//==========================================================
// 8) Extend automatic unload pulses
//==========================================================
// EN: A 500 ms pulse is compatible with integrated and third-party stackers.
// PT: Um pulso de 500 ms é compatível com stackers integrados e de terceiros.
instTPUpperStackerUnload(
    IN := upperStackerUnload,
    PT := T#500MS
);

instTPLowerStackerUnload(
    IN := lowerStackerUnload,
    PT := T#500MS
);

upperStackerUnload := instTPUpperStackerUnload.Q;
lowerStackerUnload := instTPLowerStackerUnload.Q;
END_ACTION

END_FUNCTION_BLOCK

// ---- POUs/MAIN.TcPOU
PROGRAM MAIN
VAR
	//==============================================================
	// EN: Main machine control function blocks
	// PT: Blocos principais de controle da máquina
	//==============================================================
	instFBSlitter1Control              : FB_SlitterControl;
	instFB_RotaryKnife                 : FB_RotaryKnife;
	// instFB_MetricsAndCalculation    : FB_MetricsAndCalculation;
	instFB_PaperDirectionControl       : FB_PaperDirectionControl;
	instFB_AutomaticOrderChange_V1     : FB_AutomaticOrderChange_V1;
	instFB_AlarmControl                : FB_AlarmControl;
	instFBSavePersistentData           : FB_SavePersistentData;

	//==============================================================
	// EN: Stacker control function blocks
	// PT: Blocos de controle dos empilhadores
	//==============================================================
	instFBLowerStackerControl          : FB_SimpleSheetStackerControl;
	instFBLowerStackerControlV1        : FB_SimpleSheetStackerControl_1;
	instFBUpperStackerControl          : FB_ComplexSheetStackerControl;

	//==============================================================
	// EN: Persistent data control status
	// PT: Estado do controle de dados persistentes
	//==============================================================
	bStart                             : BOOL;
	bError                             : BOOL;
	bBusy                              : BOOL;
	nErrorId                           : UDINT;
	fbR_Trig                           : R_TRIG;

	//==============================================================
	// EN: Machine interlock and control signals
	// PT: Sinais de intertravamento e controle da máquina
	//==============================================================
	slitterHomeComplete                : BOOL;
	aocReferenceSwitch                 : BOOL;
	lineSpeedUpFromAOC                 : BOOL;
	lineSpeedDownFromAOC               : BOOL;
	lineStopFromAOC                    : BOOL;
	executePositioningFromAOC          : BOOL;
	rotaryKnifeSpeedRefFromAOC         : LREAL;
	slitterSpeedRefFromAOC             : LREAL;
	lineStopFromRotaryKnife            : BOOL;
	lineStopFromSlitter                : BOOL;
	lineStopFromLowerStacker           : BOOL;
	aocRunning                         : BOOL;

	//==============================================================
	// EN: Program initialization
	// PT: Inicialização do programa
	//==============================================================
	firstScan                          : BOOL := TRUE;
	lineStopFromUpperStacker: BOOL;
END_VAR

//==============================================================
// EN: Cyclic machine control sequence
// PT: Sequência cíclica de controle da máquina
//==============================================================
_00_UpdateHardware();
_01_SlitterControl();
_02_RotaryKnifeControl();
_04_AutomaticOrderChange();
_05_LineControl();
_06_AlarmsControl();
_07_LowerStackerControl();
_08_UpperStackerControl();

// EN: Publish the upper stacker alarms and include them in the general indication.
// PT: Publica os alarmes do stacker superior e os inclui na indicação geral.
hmiAlarms.upperStacker :=
	instFBUpperStackerControl.hmiAlarms;

hmiStatus.alarmActive :=
	hmiStatus.alarmActive OR
	instFBUpperStackerControl.alarmActive;

// EN: Update persistent data management.
// PT: Atualiza o gerenciamento dos dados persistentes.
instFBSavePersistentData();

// EN: Apply default commands during the first PLC scan.
// PT: Aplica os comandos padrão durante o primeiro ciclo do PLC.
IF firstScan THEN
	hmiCommands.lowerStacker.backstopAutoCmd := TRUE;
	hmiCommands.lowerStacker.conveyorLevelerAutoCmd := TRUE;

	hmiCommands.upperStacker.backstopAutoCmd := TRUE;
	hmiCommands.upperStacker.elevatorAutoCmd := TRUE;

END_IF

firstScan := FALSE;

(*==============================================================================================================================
CPNTeck - Automação industrial
(c)Copyright 2023 All Rights Reserved
_______________________________________________________________________________________________________________________________
Library: <N/A or library name>
Tested with: <PLC / IPC model>
Engineering: <TwinCAT version>
Restrictions: <text>
Requirements: <text>
Functionality: <short description>
Support: <email>
Note: Parameter comments are only available in language 'English (United States)'
_______________________________________________________________________________________________________________________________
Change log table:

Version  		| Date        			| Expert in charge  	| Changes applied
<xx.xx.xx>		| <dd.mm.yyyy>  		| <name>              | <changes>

===============================================================================================================================*)

METHOD _00_UpdateHardware
VAR_INPUT
END_VAR

SLT1_P1_100_UG1();
SLT1_P1_100_UG2();
SLT1_P1_100_UG3();
SLT1_P1_100_UG4();
SLT1_P1_100_UG5();

SLT1_P1_200_UG1();
SLT1_P1_200_UG2();
SLT1_P1_200_UG3();
SLT1_P1_200_UG4();
SLT1_P1_200_UG5();
SLT1_P1_200_UG6();
SLT1_P1_200_UG7();
SLT1_P1_200_UG8();


STK_P2_050_DI1();
STK_P2_050_DI2();
STK_P2_050_DO1();
STK_P2_050_DO2();
	
STK_P2_050_AO1();	
STK_P2_050_AO2();
STK_P2_050_AO3();
STK_P2_050_AO4();

STK_P2_050_ENC1();
//Io-Link master
STK_050_BC2();
//Io-Link Slaves

STKU_050_DIO1();	//Ch 0 - IO-Link IP67 Input/Output module
STKU_050_DIO2(); //Ch 1 - IO-Link DIN Rail Input/Output module
STKU_050_DIO3(); //Ch 1 - IO-Link DIN Rail Input/Output module


STKL_050_DIO1();	//Ch 0 - IO-Link IP67 Input/Output module
STKL_050_DIO2(); //Ch 1 - IO-Link DIN Rail Input/Output module
STKL_100_B01(); //Ch 2 - IO-Link Pile height sensor	

//CANOpen slave	
STKU_P2_100_UG8(enable := TRUE); //Backstop servo drive

// EN: Lift servo drive. Quick stop is generated by the elevator control block.
// PT: Servo do elevador. O quick stop é gerado pelo bloco de controle do elevador.
STKU_P2_100_UG9(enable := TRUE);

// Safety processor (TwinSAFE)
STK_P2_050_SP01(run := TRUE,
				 errorAcknowledgement := hmiCommands.slitter1.resetCmd OR hmiCommands.lowerStacker.resetCmd OR hmiCommands.upperStacker.resetCmd,
				 safetyReset := hmiCommands.slitter1.resetCmd OR hmiCommands.lowerStacker.resetCmd OR hmiCommands.upperStacker.resetCmd
);
END_METHOD

METHOD _01_SlitterControl
VAR_INPUT
END_VAR

//ARK_P1_050_AO02.Channel1
//ARK_P1_050_AO02.Channel3
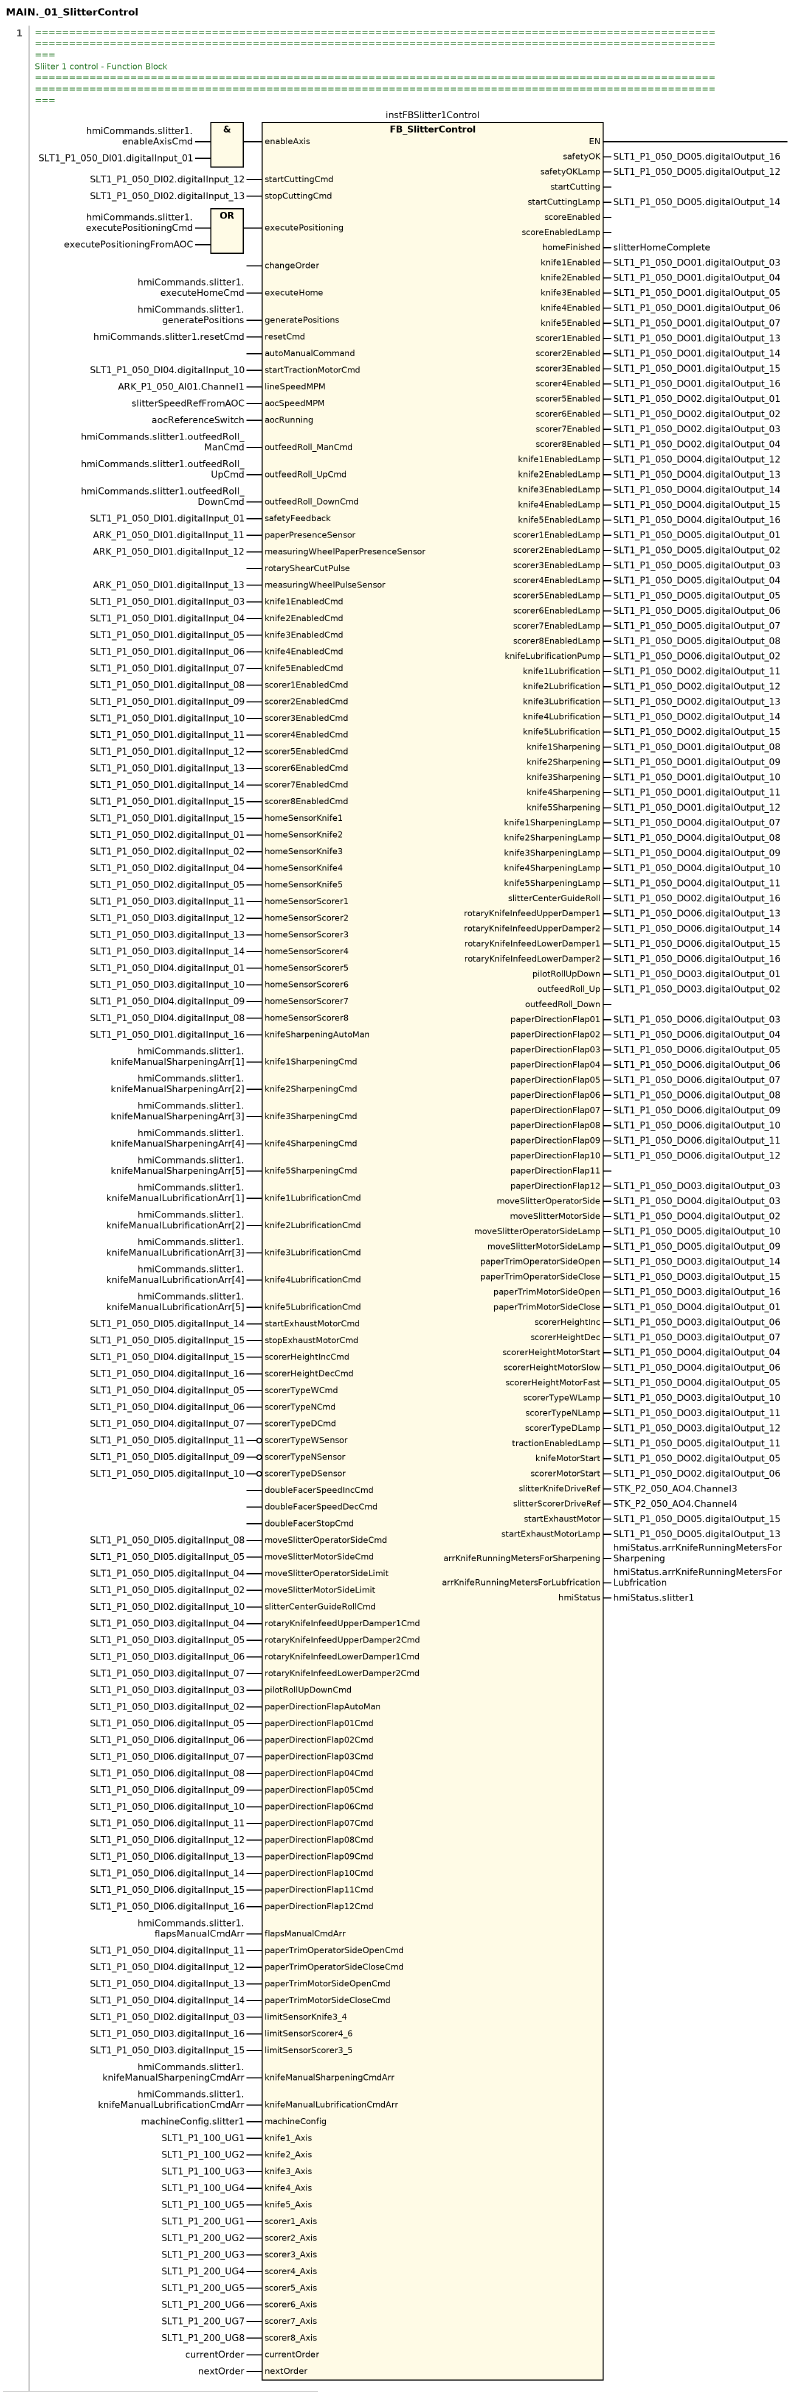
// NETWORK 1
// 					===========================================================================================================================================================================================================
//
// Sliiter 1 control - Function Block
//
// ===========================================================================================================================================================================================================
//
instFBSlitter1Control(
    enableAxis := hmiCommands.slitter1.enableAxisCmd AND SLT1_P1_050_DI01.digitalInput_01,
    startCuttingCmd := SLT1_P1_050_DI02.digitalInput_12,
    stopCuttingCmd := SLT1_P1_050_DI02.digitalInput_13,
    executePositioning := hmiCommands.slitter1.executePositioningCmd OR executePositioningFromAOC,
    executeHome := hmiCommands.slitter1.executeHomeCmd,
    generatePositions := hmiCommands.slitter1.generatePositions,
    resetCmd := hmiCommands.slitter1.resetCmd,
    startTractionMotorCmd := SLT1_P1_050_DI04.digitalInput_10,
    lineSpeedMPM := ARK_P1_050_AI01.Channel1,
    aocSpeedMPM := slitterSpeedRefFromAOC,
    aocRunning := aocReferenceSwitch,
    outfeedRoll_ManCmd := hmiCommands.slitter1.outfeedRoll_ManCmd,
    outfeedRoll_UpCmd := hmiCommands.slitter1.outfeedRoll_UpCmd,
    outfeedRoll_DownCmd := hmiCommands.slitter1.outfeedRoll_DownCmd,
    safetyFeedback := SLT1_P1_050_DI01.digitalInput_01,
    paperPresenceSensor := ARK_P1_050_DI01.digitalInput_11,
    measuringWheelPaperPresenceSensor := ARK_P1_050_DI01.digitalInput_12,
    measuringWheelPulseSensor := ARK_P1_050_DI01.digitalInput_13,
    knife1EnabledCmd := SLT1_P1_050_DI01.digitalInput_03,
    knife2EnabledCmd := SLT1_P1_050_DI01.digitalInput_04,
    knife3EnabledCmd := SLT1_P1_050_DI01.digitalInput_05,
    knife4EnabledCmd := SLT1_P1_050_DI01.digitalInput_06,
    knife5EnabledCmd := SLT1_P1_050_DI01.digitalInput_07,
    scorer1EnabledCmd := SLT1_P1_050_DI01.digitalInput_08,
    scorer2EnabledCmd := SLT1_P1_050_DI01.digitalInput_09,
    scorer3EnabledCmd := SLT1_P1_050_DI01.digitalInput_10,
    scorer4EnabledCmd := SLT1_P1_050_DI01.digitalInput_11,
    scorer5EnabledCmd := SLT1_P1_050_DI01.digitalInput_12,
    scorer6EnabledCmd := SLT1_P1_050_DI01.digitalInput_13,
    scorer7EnabledCmd := SLT1_P1_050_DI01.digitalInput_14,
    scorer8EnabledCmd := SLT1_P1_050_DI01.digitalInput_15,
    homeSensorKnife1 := SLT1_P1_050_DI01.digitalInput_15,
    homeSensorKnife2 := SLT1_P1_050_DI02.digitalInput_01,
    homeSensorKnife3 := SLT1_P1_050_DI02.digitalInput_02,
    homeSensorKnife4 := SLT1_P1_050_DI02.digitalInput_04,
    homeSensorKnife5 := SLT1_P1_050_DI02.digitalInput_05,
    homeSensorScorer1 := SLT1_P1_050_DI03.digitalInput_11,
    homeSensorScorer2 := SLT1_P1_050_DI03.digitalInput_12,
    homeSensorScorer3 := SLT1_P1_050_DI03.digitalInput_13,
    homeSensorScorer4 := SLT1_P1_050_DI03.digitalInput_14,
    homeSensorScorer5 := SLT1_P1_050_DI04.digitalInput_01,
    homeSensorScorer6 := SLT1_P1_050_DI03.digitalInput_10,
    homeSensorScorer7 := SLT1_P1_050_DI04.digitalInput_09,
    homeSensorScorer8 := SLT1_P1_050_DI04.digitalInput_08,
    knifeSharpeningAutoMan := SLT1_P1_050_DI01.digitalInput_16,
    knife1SharpeningCmd := hmiCommands.slitter1.knifeManualSharpeningArr[1],
    knife2SharpeningCmd := hmiCommands.slitter1.knifeManualSharpeningArr[2],
    knife3SharpeningCmd := hmiCommands.slitter1.knifeManualSharpeningArr[3],
    knife4SharpeningCmd := hmiCommands.slitter1.knifeManualSharpeningArr[4],
    knife5SharpeningCmd := hmiCommands.slitter1.knifeManualSharpeningArr[5],
    knife1LubrificationCmd := hmiCommands.slitter1.knifeManualLubrificationArr[1],
    knife2LubrificationCmd := hmiCommands.slitter1.knifeManualLubrificationArr[2],
    knife3LubrificationCmd := hmiCommands.slitter1.knifeManualLubrificationArr[3],
    knife4LubrificationCmd := hmiCommands.slitter1.knifeManualLubrificationArr[4],
    knife5LubrificationCmd := hmiCommands.slitter1.knifeManualLubrificationArr[5],
    startExhaustMotorCmd := SLT1_P1_050_DI05.digitalInput_14,
    stopExhaustMotorCmd := SLT1_P1_050_DI05.digitalInput_15,
    scorerHeightIncCmd := SLT1_P1_050_DI04.digitalInput_15,
    scorerHeightDecCmd := SLT1_P1_050_DI04.digitalInput_16,
    scorerTypeWCmd := SLT1_P1_050_DI04.digitalInput_05,
    scorerTypeNCmd := SLT1_P1_050_DI04.digitalInput_06,
    scorerTypeDCmd := SLT1_P1_050_DI04.digitalInput_07,
    scorerTypeWSensor := NOT SLT1_P1_050_DI05.digitalInput_11,
    scorerTypeNSensor := NOT SLT1_P1_050_DI05.digitalInput_09,
    scorerTypeDSensor := NOT SLT1_P1_050_DI05.digitalInput_10,
    moveSlitterOperatorSideCmd := SLT1_P1_050_DI05.digitalInput_08,
    moveSlitterMotorSideCmd := SLT1_P1_050_DI05.digitalInput_05,
    moveSlitterOperatorSideLimit := SLT1_P1_050_DI05.digitalInput_04,
    moveSlitterMotorSideLimit := SLT1_P1_050_DI05.digitalInput_02,
    slitterCenterGuideRollCmd := SLT1_P1_050_DI02.digitalInput_10,
    rotaryKnifeInfeedUpperDamper1Cmd := SLT1_P1_050_DI03.digitalInput_04,
    rotaryKnifeInfeedUpperDamper2Cmd := SLT1_P1_050_DI03.digitalInput_05,
    rotaryKnifeInfeedLowerDamper1Cmd := SLT1_P1_050_DI03.digitalInput_06,
    rotaryKnifeInfeedLowerDamper2Cmd := SLT1_P1_050_DI03.digitalInput_07,
    pilotRollUpDownCmd := SLT1_P1_050_DI03.digitalInput_03,
    paperDirectionFlapAutoMan := SLT1_P1_050_DI03.digitalInput_02,
    paperDirectionFlap01Cmd := SLT1_P1_050_DI06.digitalInput_05,
    paperDirectionFlap02Cmd := SLT1_P1_050_DI06.digitalInput_06,
    paperDirectionFlap03Cmd := SLT1_P1_050_DI06.digitalInput_07,
    paperDirectionFlap04Cmd := SLT1_P1_050_DI06.digitalInput_08,
    paperDirectionFlap05Cmd := SLT1_P1_050_DI06.digitalInput_09,
    paperDirectionFlap06Cmd := SLT1_P1_050_DI06.digitalInput_10,
    paperDirectionFlap07Cmd := SLT1_P1_050_DI06.digitalInput_11,
    paperDirectionFlap08Cmd := SLT1_P1_050_DI06.digitalInput_12,
    paperDirectionFlap09Cmd := SLT1_P1_050_DI06.digitalInput_13,
    paperDirectionFlap10Cmd := SLT1_P1_050_DI06.digitalInput_14,
    paperDirectionFlap11Cmd := SLT1_P1_050_DI06.digitalInput_15,
    paperDirectionFlap12Cmd := SLT1_P1_050_DI06.digitalInput_16,
    flapsManualCmdArr := hmiCommands.slitter1.flapsManualCmdArr,
    paperTrimOperatorSideOpenCmd := SLT1_P1_050_DI04.digitalInput_11,
    paperTrimOperatorSideCloseCmd := SLT1_P1_050_DI04.digitalInput_12,
    paperTrimMotorSideOpenCmd := SLT1_P1_050_DI04.digitalInput_13,
    paperTrimMotorSideCloseCmd := SLT1_P1_050_DI04.digitalInput_14,
    limitSensorKnife3_4 := SLT1_P1_050_DI02.digitalInput_03,
    limitSensorScorer4_6 := SLT1_P1_050_DI03.digitalInput_16,
    limitSensorScorer3_5 := SLT1_P1_050_DI03.digitalInput_15,
    knifeManualSharpeningCmdArr := hmiCommands.slitter1.knifeManualSharpeningCmdArr,
    knifeManualLubrificationCmdArr := hmiCommands.slitter1.knifeManualLubrificationCmdArr,
    machineConfig := machineConfig.slitter1,
    knife1_Axis := SLT1_P1_100_UG1,
    knife2_Axis := SLT1_P1_100_UG2,
    knife3_Axis := SLT1_P1_100_UG3,
    knife4_Axis := SLT1_P1_100_UG4,
    knife5_Axis := SLT1_P1_100_UG5,
    scorer1_Axis := SLT1_P1_200_UG1,
    scorer2_Axis := SLT1_P1_200_UG2,
    scorer3_Axis := SLT1_P1_200_UG3,
    scorer4_Axis := SLT1_P1_200_UG4,
    scorer5_Axis := SLT1_P1_200_UG5,
    scorer6_Axis := SLT1_P1_200_UG6,
    scorer7_Axis := SLT1_P1_200_UG7,
    scorer8_Axis := SLT1_P1_200_UG8,
    currentOrder := currentOrder,
    nextOrder := nextOrder,
    safetyOK => SLT1_P1_050_DO05.digitalOutput_16,
    safetyOKLamp => SLT1_P1_050_DO05.digitalOutput_12,
    startCuttingLamp => SLT1_P1_050_DO05.digitalOutput_14,
    homeFinished => slitterHomeComplete,
    knife1Enabled => SLT1_P1_050_DO01.digitalOutput_03,
    knife2Enabled => SLT1_P1_050_DO01.digitalOutput_04,
    knife3Enabled => SLT1_P1_050_DO01.digitalOutput_05,
    knife4Enabled => SLT1_P1_050_DO01.digitalOutput_06,
    knife5Enabled => SLT1_P1_050_DO01.digitalOutput_07,
    scorer1Enabled => SLT1_P1_050_DO01.digitalOutput_13,
    scorer2Enabled => SLT1_P1_050_DO01.digitalOutput_14,
    scorer3Enabled => SLT1_P1_050_DO01.digitalOutput_15,
    scorer4Enabled => SLT1_P1_050_DO01.digitalOutput_16,
    scorer5Enabled => SLT1_P1_050_DO02.digitalOutput_01,
    scorer6Enabled => SLT1_P1_050_DO02.digitalOutput_02,
    scorer7Enabled => SLT1_P1_050_DO02.digitalOutput_03,
    scorer8Enabled => SLT1_P1_050_DO02.digitalOutput_04,
    knife1EnabledLamp => SLT1_P1_050_DO04.digitalOutput_12,
    knife2EnabledLamp => SLT1_P1_050_DO04.digitalOutput_13,
    knife3EnabledLamp => SLT1_P1_050_DO04.digitalOutput_14,
    knife4EnabledLamp => SLT1_P1_050_DO04.digitalOutput_15,
    knife5EnabledLamp => SLT1_P1_050_DO04.digitalOutput_16,
    scorer1EnabledLamp => SLT1_P1_050_DO05.digitalOutput_01,
    scorer2EnabledLamp => SLT1_P1_050_DO05.digitalOutput_02,
    scorer3EnabledLamp => SLT1_P1_050_DO05.digitalOutput_03,
    scorer4EnabledLamp => SLT1_P1_050_DO05.digitalOutput_04,
    scorer5EnabledLamp => SLT1_P1_050_DO05.digitalOutput_05,
    scorer6EnabledLamp => SLT1_P1_050_DO05.digitalOutput_06,
    scorer7EnabledLamp => SLT1_P1_050_DO05.digitalOutput_07,
    scorer8EnabledLamp => SLT1_P1_050_DO05.digitalOutput_08,
    knifeLubrificationPump => SLT1_P1_050_DO06.digitalOutput_02,
    knife1Lubrification => SLT1_P1_050_DO02.digitalOutput_11,
    knife2Lubrification => SLT1_P1_050_DO02.digitalOutput_12,
    knife3Lubrification => SLT1_P1_050_DO02.digitalOutput_13,
    knife4Lubrification => SLT1_P1_050_DO02.digitalOutput_14,
    knife5Lubrification => SLT1_P1_050_DO02.digitalOutput_15,
    knife1Sharpening => SLT1_P1_050_DO01.digitalOutput_08,
    knife2Sharpening => SLT1_P1_050_DO01.digitalOutput_09,
    knife3Sharpening => SLT1_P1_050_DO01.digitalOutput_10,
    knife4Sharpening => SLT1_P1_050_DO01.digitalOutput_11,
    knife5Sharpening => SLT1_P1_050_DO01.digitalOutput_12,
    knife1SharpeningLamp => SLT1_P1_050_DO04.digitalOutput_07,
    knife2SharpeningLamp => SLT1_P1_050_DO04.digitalOutput_08,
    knife3SharpeningLamp => SLT1_P1_050_DO04.digitalOutput_09,
    knife4SharpeningLamp => SLT1_P1_050_DO04.digitalOutput_10,
    knife5SharpeningLamp => SLT1_P1_050_DO04.digitalOutput_11,
    slitterCenterGuideRoll => SLT1_P1_050_DO02.digitalOutput_16,
    rotaryKnifeInfeedUpperDamper1 => SLT1_P1_050_DO06.digitalOutput_13,
    rotaryKnifeInfeedUpperDamper2 => SLT1_P1_050_DO06.digitalOutput_14,
    rotaryKnifeInfeedLowerDamper1 => SLT1_P1_050_DO06.digitalOutput_15,
    rotaryKnifeInfeedLowerDamper2 => SLT1_P1_050_DO06.digitalOutput_16,
    pilotRollUpDown => SLT1_P1_050_DO03.digitalOutput_01,
    outfeedRoll_Up => SLT1_P1_050_DO03.digitalOutput_02,
    paperDirectionFlap01 => SLT1_P1_050_DO06.digitalOutput_03,
    paperDirectionFlap02 => SLT1_P1_050_DO06.digitalOutput_04,
    paperDirectionFlap03 => SLT1_P1_050_DO06.digitalOutput_05,
    paperDirectionFlap04 => SLT1_P1_050_DO06.digitalOutput_06,
    paperDirectionFlap05 => SLT1_P1_050_DO06.digitalOutput_07,
    paperDirectionFlap06 => SLT1_P1_050_DO06.digitalOutput_08,
    paperDirectionFlap07 => SLT1_P1_050_DO06.digitalOutput_09,
    paperDirectionFlap08 => SLT1_P1_050_DO06.digitalOutput_10,
    paperDirectionFlap09 => SLT1_P1_050_DO06.digitalOutput_11,
    paperDirectionFlap10 => SLT1_P1_050_DO06.digitalOutput_12,
    paperDirectionFlap12 => SLT1_P1_050_DO03.digitalOutput_03,
    moveSlitterOperatorSide => SLT1_P1_050_DO04.digitalOutput_03,
    moveSlitterMotorSide => SLT1_P1_050_DO04.digitalOutput_02,
    moveSlitterOperatorSideLamp => SLT1_P1_050_DO05.digitalOutput_10,
    moveSlitterMotorSideLamp => SLT1_P1_050_DO05.digitalOutput_09,
    paperTrimOperatorSideOpen => SLT1_P1_050_DO03.digitalOutput_14,
    paperTrimOperatorSideClose => SLT1_P1_050_DO03.digitalOutput_15,
    paperTrimMotorSideOpen => SLT1_P1_050_DO03.digitalOutput_16,
    paperTrimMotorSideClose => SLT1_P1_050_DO04.digitalOutput_01,
    scorerHeightInc => SLT1_P1_050_DO03.digitalOutput_06,
    scorerHeightDec => SLT1_P1_050_DO03.digitalOutput_07,
    scorerHeightMotorStart => SLT1_P1_050_DO04.digitalOutput_04,
    scorerHeightMotorSlow => SLT1_P1_050_DO04.digitalOutput_06,
    scorerHeightMotorFast => SLT1_P1_050_DO04.digitalOutput_05,
    scorerTypeWLamp => SLT1_P1_050_DO03.digitalOutput_10,
    scorerTypeNLamp => SLT1_P1_050_DO03.digitalOutput_11,
    scorerTypeDLamp => SLT1_P1_050_DO03.digitalOutput_12,
    tractionEnabledLamp => SLT1_P1_050_DO05.digitalOutput_11,
    knifeMotorStart => SLT1_P1_050_DO02.digitalOutput_05,
    scorerMotorStart => SLT1_P1_050_DO02.digitalOutput_06,
    slitterKnifeDriveRef => STK_P2_050_AO4.Channel3,
    slitterScorerDriveRef => STK_P2_050_AO4.Channel4,
    startExhaustMotor => SLT1_P1_050_DO05.digitalOutput_15,
    startExhaustMotorLamp => SLT1_P1_050_DO05.digitalOutput_13,
    arrKnifeRunningMetersForSharpening => hmiStatus.arrKnifeRunningMetersForSharpening,
    arrKnifeRunningMetersForLubfrication => hmiStatus.arrKnifeRunningMetersForLubfrication,
    hmiStatus => hmiStatus.slitter1); // FB_SlitterControl
END_METHOD

METHOD _02_RotaryKnifeControl
VAR_INPUT
END_VAR

(*


ARK_050_DI01.digitalInput_01 => exitGuardOpen
ARK_050_DI01.digitalInput_02 => lowerKnifeGuardClosed
ARK_050_DI01.digitalInput_03 => upperKnifeGuardClosed
ARK_050_DI01.digitalInput_04 => infeedGuardOpen

ARK_050_DI01.digitalInput_05 => lowerOilLevelLow
ARK_050_DI01.digitalInput_06 => upperOilLevelLow
ARK_050_DI01.digitalInput_07 => exhaustPressurized
ARK_050_DI01.digitalInput_08 => exhaustDepressurized

ARK_050_DI01.digitalInput_09 => upperLevelPaperSensor
ARK_050_DI01.digitalInput_10 => upperKnifeJamDetected
ARK_050_DI01.digitalInput_11 => lowerLevelPaperSensor
ARK_050_DI01.digitalInput_12 => lowerKnifeJamDetected

ARK_050_DI01.digitalInput_13 => lowerKnifeHome
ARK_050_DI01.digitalInput_14 => upperKnifeHome

*)
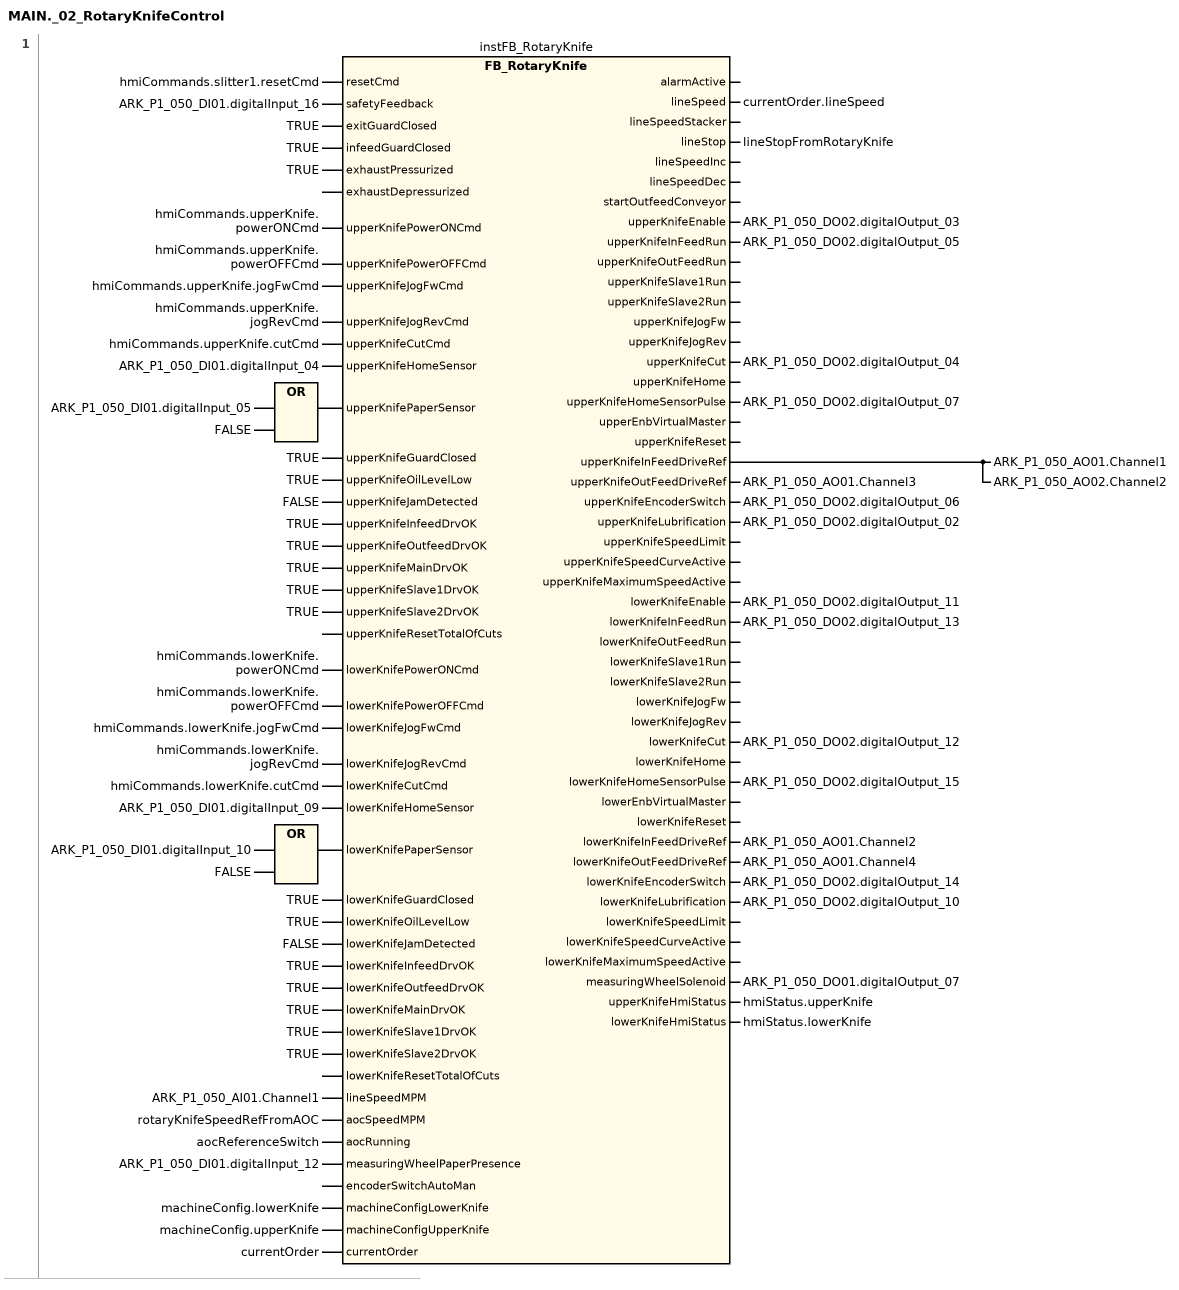
// NETWORK 1
instFB_RotaryKnife(
    resetCmd := hmiCommands.slitter1.resetCmd,
    safetyFeedback := ARK_P1_050_DI01.digitalInput_16,
    exitGuardClosed := TRUE,
    infeedGuardClosed := TRUE,
    exhaustPressurized := TRUE,
    upperKnifePowerONCmd := hmiCommands.upperKnife.powerONCmd,
    upperKnifePowerOFFCmd := hmiCommands.upperKnife.powerOFFCmd,
    upperKnifeJogFwCmd := hmiCommands.upperKnife.jogFwCmd,
    upperKnifeJogRevCmd := hmiCommands.upperKnife.jogRevCmd,
    upperKnifeCutCmd := hmiCommands.upperKnife.cutCmd,
    upperKnifeHomeSensor := ARK_P1_050_DI01.digitalInput_04,
    upperKnifePaperSensor := ARK_P1_050_DI01.digitalInput_05 OR FALSE,
    upperKnifeGuardClosed := TRUE,
    upperKnifeOilLevelLow := TRUE,
    upperKnifeJamDetected := FALSE,
    upperKnifeInfeedDrvOK := TRUE,
    upperKnifeOutfeedDrvOK := TRUE,
    upperKnifeMainDrvOK := TRUE,
    upperKnifeSlave1DrvOK := TRUE,
    upperKnifeSlave2DrvOK := TRUE,
    lowerKnifePowerONCmd := hmiCommands.lowerKnife.powerONCmd,
    lowerKnifePowerOFFCmd := hmiCommands.lowerKnife.powerOFFCmd,
    lowerKnifeJogFwCmd := hmiCommands.lowerKnife.jogFwCmd,
    lowerKnifeJogRevCmd := hmiCommands.lowerKnife.jogRevCmd,
    lowerKnifeCutCmd := hmiCommands.lowerKnife.cutCmd,
    lowerKnifeHomeSensor := ARK_P1_050_DI01.digitalInput_09,
    lowerKnifePaperSensor := ARK_P1_050_DI01.digitalInput_10 OR FALSE,
    lowerKnifeGuardClosed := TRUE,
    lowerKnifeOilLevelLow := TRUE,
    lowerKnifeJamDetected := FALSE,
    lowerKnifeInfeedDrvOK := TRUE,
    lowerKnifeOutfeedDrvOK := TRUE,
    lowerKnifeMainDrvOK := TRUE,
    lowerKnifeSlave1DrvOK := TRUE,
    lowerKnifeSlave2DrvOK := TRUE,
    lineSpeedMPM := ARK_P1_050_AI01.Channel1,
    aocSpeedMPM := rotaryKnifeSpeedRefFromAOC,
    aocRunning := aocReferenceSwitch,
    measuringWheelPaperPresence := ARK_P1_050_DI01.digitalInput_12,
    machineConfigLowerKnife := machineConfig.lowerKnife,
    machineConfigUpperKnife := machineConfig.upperKnife,
    currentOrder := currentOrder,
    lineSpeed => currentOrder.lineSpeed,
    lineStop => lineStopFromRotaryKnife,
    upperKnifeEnable => ARK_P1_050_DO02.digitalOutput_03,
    upperKnifeInFeedRun => ARK_P1_050_DO02.digitalOutput_05,
    upperKnifeCut => ARK_P1_050_DO02.digitalOutput_04,
    upperKnifeHomeSensorPulse => ARK_P1_050_DO02.digitalOutput_07,
    upperKnifeOutFeedDriveRef => ARK_P1_050_AO01.Channel3,
    upperKnifeEncoderSwitch => ARK_P1_050_DO02.digitalOutput_06,
    upperKnifeLubrification => ARK_P1_050_DO02.digitalOutput_02,
    lowerKnifeEnable => ARK_P1_050_DO02.digitalOutput_11,
    lowerKnifeInFeedRun => ARK_P1_050_DO02.digitalOutput_13,
    lowerKnifeCut => ARK_P1_050_DO02.digitalOutput_12,
    lowerKnifeHomeSensorPulse => ARK_P1_050_DO02.digitalOutput_15,
    lowerKnifeInFeedDriveRef => ARK_P1_050_AO01.Channel2,
    lowerKnifeOutFeedDriveRef => ARK_P1_050_AO01.Channel4,
    lowerKnifeEncoderSwitch => ARK_P1_050_DO02.digitalOutput_14,
    lowerKnifeLubrification => ARK_P1_050_DO02.digitalOutput_10,
    measuringWheelSolenoid => ARK_P1_050_DO01.digitalOutput_07,
    upperKnifeHmiStatus => hmiStatus.upperKnife,
    lowerKnifeHmiStatus => hmiStatus.lowerKnife); // FB_RotaryKnife
ARK_P1_050_AO01.Channel1 := instFB_RotaryKnife.upperKnifeInFeedDriveRef;
ARK_P1_050_AO02.Channel2 := instFB_RotaryKnife.upperKnifeInFeedDriveRef;
END_METHOD

METHOD _04_AutomaticOrderChange
VAR_INPUT
END_VAR
(*

	SLT1_C1_050_DI01     : FB_EL1809;        // Digital inputs card
    SLT1_C1_050_DO01     : FB_EL2809;        // Digital outputs card

*)
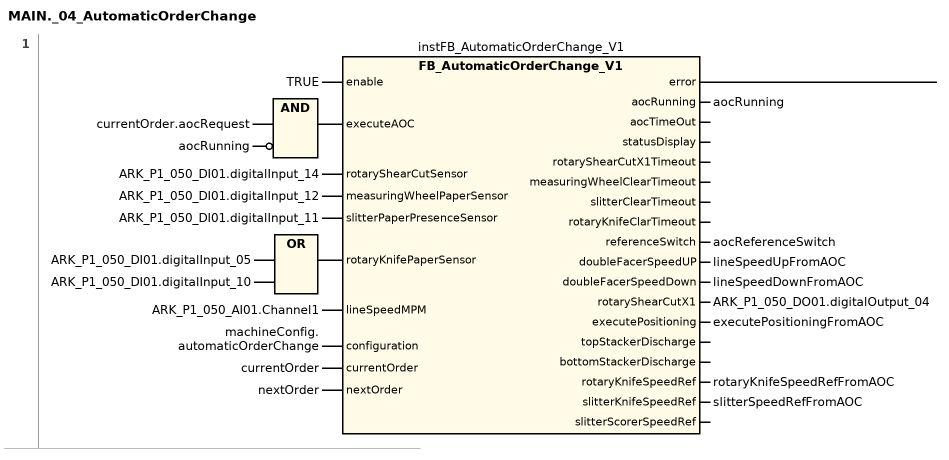
// NETWORK 1
instFB_AutomaticOrderChange_V1(
    enable := TRUE,
    executeAOC := currentOrder.aocRequest AND NOT aocRunning,
    rotaryShearCutSensor := ARK_P1_050_DI01.digitalInput_14,
    measuringWheelPaperSensor := ARK_P1_050_DI01.digitalInput_12,
    slitterPaperPresenceSensor := ARK_P1_050_DI01.digitalInput_11,
    rotaryKnifePaperSensor := ARK_P1_050_DI01.digitalInput_05 OR ARK_P1_050_DI01.digitalInput_10,
    lineSpeedMPM := ARK_P1_050_AI01.Channel1,
    configuration := machineConfig.automaticOrderChange,
    currentOrder := currentOrder,
    nextOrder := nextOrder,
    aocRunning => aocRunning,
    referenceSwitch => aocReferenceSwitch,
    doubleFacerSpeedUP => lineSpeedUpFromAOC,
    doubleFacerSpeedDown => lineSpeedDownFromAOC,
    rotaryShearCutX1 => ARK_P1_050_DO01.digitalOutput_04,
    executePositioning => executePositioningFromAOC,
    rotaryKnifeSpeedRef => rotaryKnifeSpeedRefFromAOC,
    slitterKnifeSpeedRef => slitterSpeedRefFromAOC); // FB_AutomaticOrderChange_V1
END_METHOD

METHOD _05_LineControl
VAR_INPUT
END_VAR
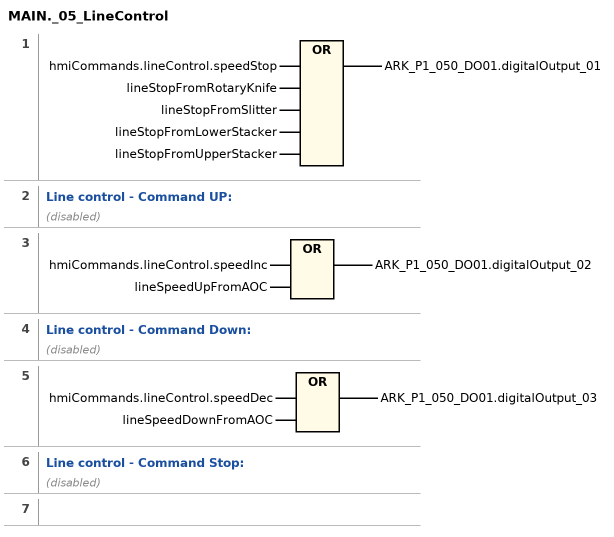
// NETWORK 1
ARK_P1_050_DO01.digitalOutput_01 := hmiCommands.lineControl.speedStop OR lineStopFromRotaryKnife OR lineStopFromSlitter OR lineStopFromLowerStacker OR lineStopFromUpperStacker;

// NETWORK 2 (disabled)
// label: Line control - Command UP

// NETWORK 3
ARK_P1_050_DO01.digitalOutput_02 := hmiCommands.lineControl.speedInc OR lineSpeedUpFromAOC;

// NETWORK 4 (disabled)
// label: Line control - Command Down

// NETWORK 5
ARK_P1_050_DO01.digitalOutput_03 := hmiCommands.lineControl.speedDec OR lineSpeedDownFromAOC;

// NETWORK 6 (disabled)
// label: Line control - Command Stop

// NETWORK 7
END_METHOD

METHOD _06_AlarmsControl
VAR_INPUT
END_VAR
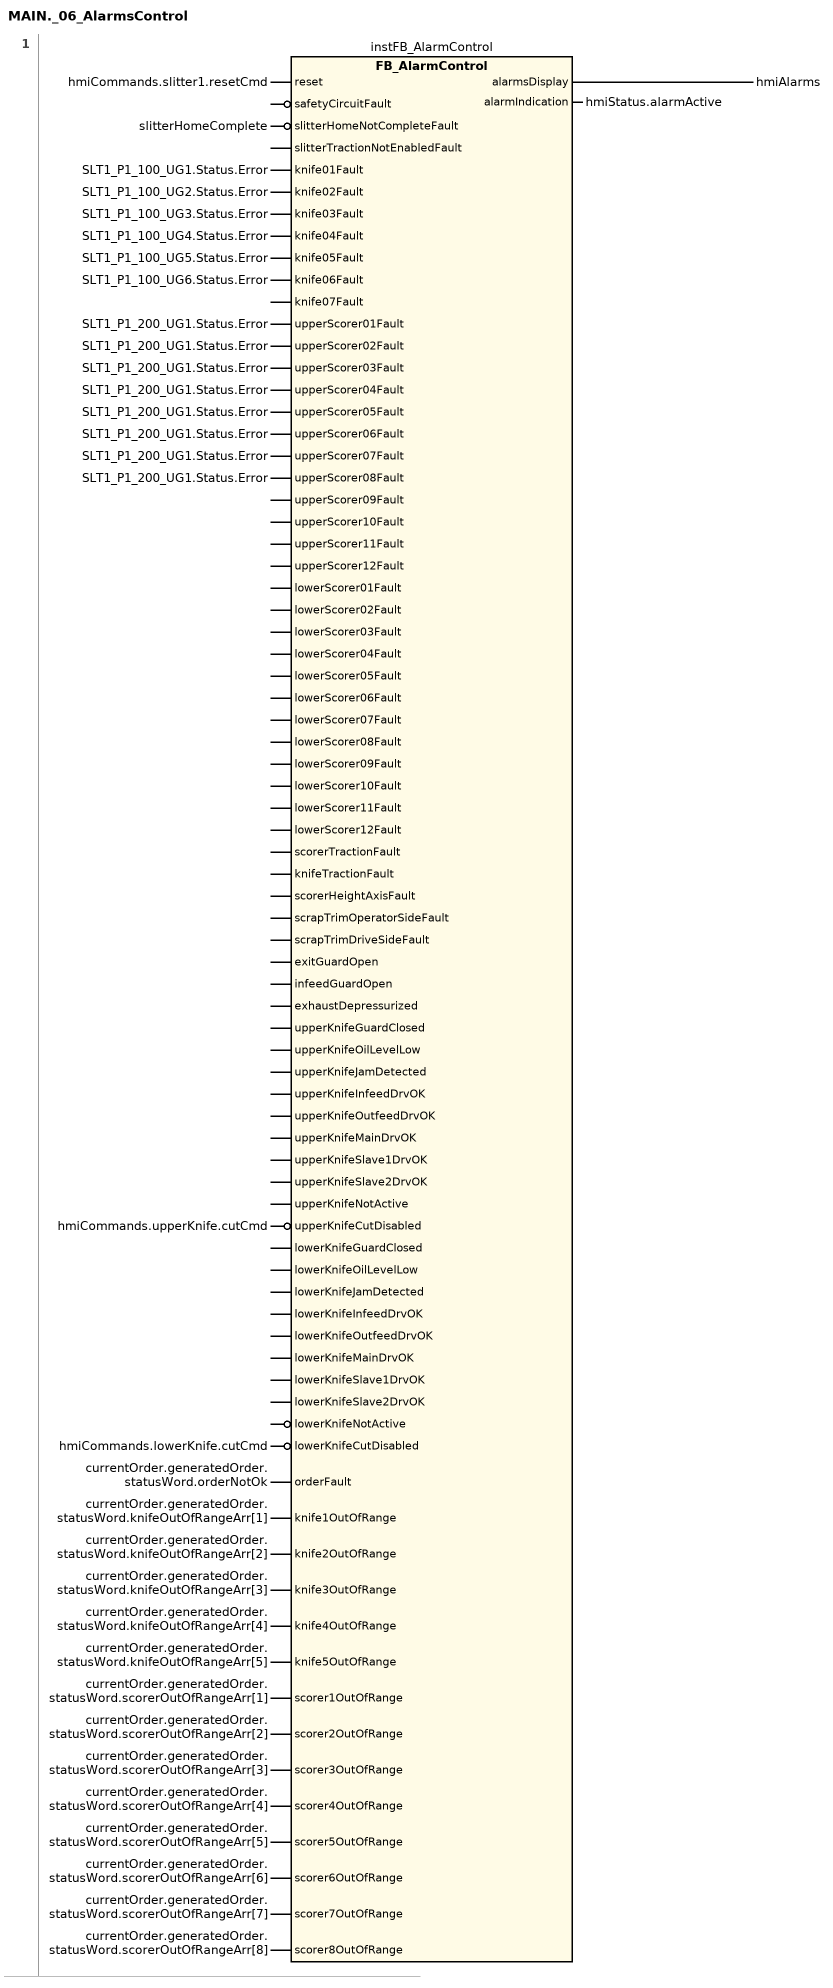
// NETWORK 1
instFB_AlarmControl(
    reset := hmiCommands.slitter1.resetCmd,
    slitterHomeNotCompleteFault := NOT slitterHomeComplete,
    knife01Fault := SLT1_P1_100_UG1.Status.Error,
    knife02Fault := SLT1_P1_100_UG2.Status.Error,
    knife03Fault := SLT1_P1_100_UG3.Status.Error,
    knife04Fault := SLT1_P1_100_UG4.Status.Error,
    knife05Fault := SLT1_P1_100_UG5.Status.Error,
    knife06Fault := SLT1_P1_100_UG6.Status.Error,
    upperScorer01Fault := SLT1_P1_200_UG1.Status.Error,
    upperScorer02Fault := SLT1_P1_200_UG1.Status.Error,
    upperScorer03Fault := SLT1_P1_200_UG1.Status.Error,
    upperScorer04Fault := SLT1_P1_200_UG1.Status.Error,
    upperScorer05Fault := SLT1_P1_200_UG1.Status.Error,
    upperScorer06Fault := SLT1_P1_200_UG1.Status.Error,
    upperScorer07Fault := SLT1_P1_200_UG1.Status.Error,
    upperScorer08Fault := SLT1_P1_200_UG1.Status.Error,
    upperKnifeCutDisabled := NOT hmiCommands.upperKnife.cutCmd,
    lowerKnifeCutDisabled := NOT hmiCommands.lowerKnife.cutCmd,
    orderFault := currentOrder.generatedOrder.statusWord.orderNotOk,
    knife1OutOfRange := currentOrder.generatedOrder.statusWord.knifeOutOfRangeArr[1],
    knife2OutOfRange := currentOrder.generatedOrder.statusWord.knifeOutOfRangeArr[2],
    knife3OutOfRange := currentOrder.generatedOrder.statusWord.knifeOutOfRangeArr[3],
    knife4OutOfRange := currentOrder.generatedOrder.statusWord.knifeOutOfRangeArr[4],
    knife5OutOfRange := currentOrder.generatedOrder.statusWord.knifeOutOfRangeArr[5],
    scorer1OutOfRange := currentOrder.generatedOrder.statusWord.scorerOutOfRangeArr[1],
    scorer2OutOfRange := currentOrder.generatedOrder.statusWord.scorerOutOfRangeArr[2],
    scorer3OutOfRange := currentOrder.generatedOrder.statusWord.scorerOutOfRangeArr[3],
    scorer4OutOfRange := currentOrder.generatedOrder.statusWord.scorerOutOfRangeArr[4],
    scorer5OutOfRange := currentOrder.generatedOrder.statusWord.scorerOutOfRangeArr[5],
    scorer6OutOfRange := currentOrder.generatedOrder.statusWord.scorerOutOfRangeArr[6],
    scorer7OutOfRange := currentOrder.generatedOrder.statusWord.scorerOutOfRangeArr[7],
    scorer8OutOfRange := currentOrder.generatedOrder.statusWord.scorerOutOfRangeArr[8],
    alarmIndication => hmiStatus.alarmActive); // FB_AlarmControl
hmiAlarms := instFB_AlarmControl.alarmsDisplay;
END_METHOD

METHOD _07_LowerStackerControl
VAR_INPUT
END_VAR

VAR
	
//ARK_P1_050_AO01.Channel2
END_VAR
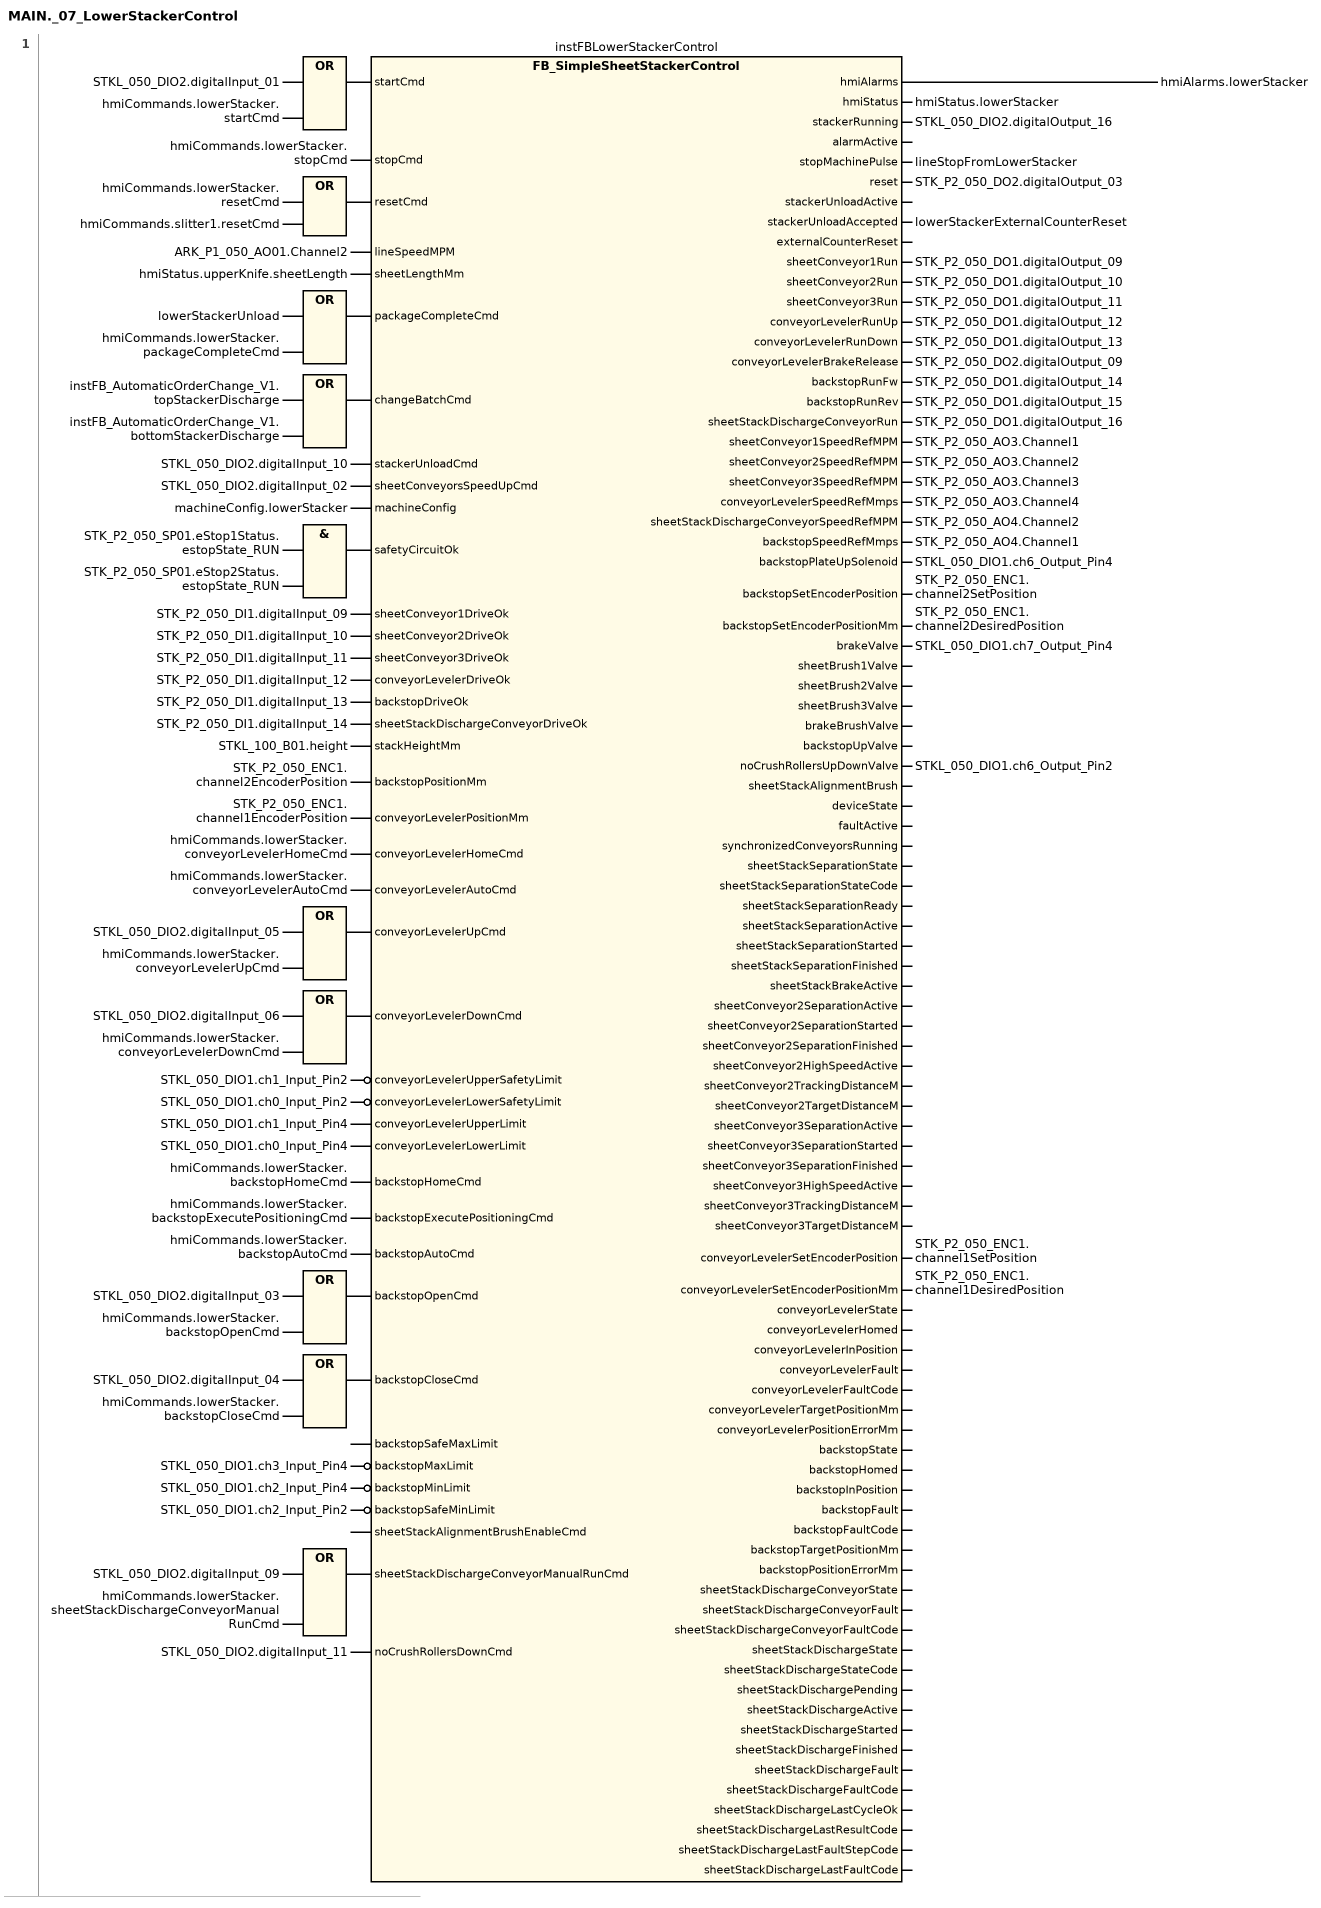
// NETWORK 1
instFBLowerStackerControl(
    startCmd := STKL_050_DIO2.digitalInput_01 OR hmiCommands.lowerStacker.startCmd,
    stopCmd := hmiCommands.lowerStacker.stopCmd,
    resetCmd := hmiCommands.lowerStacker.resetCmd OR hmiCommands.slitter1.resetCmd,
    lineSpeedMPM := ARK_P1_050_AO01.Channel2,
    sheetLengthMm := hmiStatus.upperKnife.sheetLength,
    packageCompleteCmd := lowerStackerUnload OR hmiCommands.lowerStacker.packageCompleteCmd,
    changeBatchCmd := instFB_AutomaticOrderChange_V1.topStackerDischarge OR instFB_AutomaticOrderChange_V1.bottomStackerDischarge,
    stackerUnloadCmd := STKL_050_DIO2.digitalInput_10,
    sheetConveyorsSpeedUpCmd := STKL_050_DIO2.digitalInput_02,
    machineConfig := machineConfig.lowerStacker,
    safetyCircuitOk := STK_P2_050_SP01.eStop1Status.estopState_RUN AND STK_P2_050_SP01.eStop2Status.estopState_RUN,
    sheetConveyor1DriveOk := STK_P2_050_DI1.digitalInput_09,
    sheetConveyor2DriveOk := STK_P2_050_DI1.digitalInput_10,
    sheetConveyor3DriveOk := STK_P2_050_DI1.digitalInput_11,
    conveyorLevelerDriveOk := STK_P2_050_DI1.digitalInput_12,
    backstopDriveOk := STK_P2_050_DI1.digitalInput_13,
    sheetStackDischargeConveyorDriveOk := STK_P2_050_DI1.digitalInput_14,
    stackHeightMm := STKL_100_B01.height,
    backstopPositionMm := STK_P2_050_ENC1.channel2EncoderPosition,
    conveyorLevelerPositionMm := STK_P2_050_ENC1.channel1EncoderPosition,
    conveyorLevelerHomeCmd := hmiCommands.lowerStacker.conveyorLevelerHomeCmd,
    conveyorLevelerAutoCmd := hmiCommands.lowerStacker.conveyorLevelerAutoCmd,
    conveyorLevelerUpCmd := STKL_050_DIO2.digitalInput_05 OR hmiCommands.lowerStacker.conveyorLevelerUpCmd,
    conveyorLevelerDownCmd := STKL_050_DIO2.digitalInput_06 OR hmiCommands.lowerStacker.conveyorLevelerDownCmd,
    conveyorLevelerUpperSafetyLimit := NOT STKL_050_DIO1.ch1_Input_Pin2,
    conveyorLevelerLowerSafetyLimit := NOT STKL_050_DIO1.ch0_Input_Pin2,
    conveyorLevelerUpperLimit := STKL_050_DIO1.ch1_Input_Pin4,
    conveyorLevelerLowerLimit := STKL_050_DIO1.ch0_Input_Pin4,
    backstopHomeCmd := hmiCommands.lowerStacker.backstopHomeCmd,
    backstopExecutePositioningCmd := hmiCommands.lowerStacker.backstopExecutePositioningCmd,
    backstopAutoCmd := hmiCommands.lowerStacker.backstopAutoCmd,
    backstopOpenCmd := STKL_050_DIO2.digitalInput_03 OR hmiCommands.lowerStacker.backstopOpenCmd,
    backstopCloseCmd := STKL_050_DIO2.digitalInput_04 OR hmiCommands.lowerStacker.backstopCloseCmd,
    backstopMaxLimit := NOT STKL_050_DIO1.ch3_Input_Pin4,
    backstopMinLimit := NOT STKL_050_DIO1.ch2_Input_Pin4,
    backstopSafeMinLimit := NOT STKL_050_DIO1.ch2_Input_Pin2,
    sheetStackDischargeConveyorManualRunCmd := STKL_050_DIO2.digitalInput_09 OR hmiCommands.lowerStacker.sheetStackDischargeConveyorManualRunCmd,
    noCrushRollersDownCmd := STKL_050_DIO2.digitalInput_11,
    hmiStatus => hmiStatus.lowerStacker,
    stackerRunning => STKL_050_DIO2.digitalOutput_16,
    stopMachinePulse => lineStopFromLowerStacker,
    reset => STK_P2_050_DO2.digitalOutput_03,
    stackerUnloadAccepted => lowerStackerExternalCounterReset,
    sheetConveyor1Run => STK_P2_050_DO1.digitalOutput_09,
    sheetConveyor2Run => STK_P2_050_DO1.digitalOutput_10,
    sheetConveyor3Run => STK_P2_050_DO1.digitalOutput_11,
    conveyorLevelerRunUp => STK_P2_050_DO1.digitalOutput_12,
    conveyorLevelerRunDown => STK_P2_050_DO1.digitalOutput_13,
    conveyorLevelerBrakeRelease => STK_P2_050_DO2.digitalOutput_09,
    backstopRunFw => STK_P2_050_DO1.digitalOutput_14,
    backstopRunRev => STK_P2_050_DO1.digitalOutput_15,
    sheetStackDischargeConveyorRun => STK_P2_050_DO1.digitalOutput_16,
    sheetConveyor1SpeedRefMPM => STK_P2_050_AO3.Channel1,
    sheetConveyor2SpeedRefMPM => STK_P2_050_AO3.Channel2,
    sheetConveyor3SpeedRefMPM => STK_P2_050_AO3.Channel3,
    conveyorLevelerSpeedRefMmps => STK_P2_050_AO3.Channel4,
    sheetStackDischargeConveyorSpeedRefMPM => STK_P2_050_AO4.Channel2,
    backstopSpeedRefMmps => STK_P2_050_AO4.Channel1,
    backstopPlateUpSolenoid => STKL_050_DIO1.ch6_Output_Pin4,
    backstopSetEncoderPosition => STK_P2_050_ENC1.channel2SetPosition,
    backstopSetEncoderPositionMm => STK_P2_050_ENC1.channel2DesiredPosition,
    brakeValve => STKL_050_DIO1.ch7_Output_Pin4,
    noCrushRollersUpDownValve => STKL_050_DIO1.ch6_Output_Pin2,
    conveyorLevelerSetEncoderPosition => STK_P2_050_ENC1.channel1SetPosition,
    conveyorLevelerSetEncoderPositionMm => STK_P2_050_ENC1.channel1DesiredPosition); // FB_SimpleSheetStackerControl
hmiAlarms.lowerStacker := instFBLowerStackerControl.hmiAlarms;

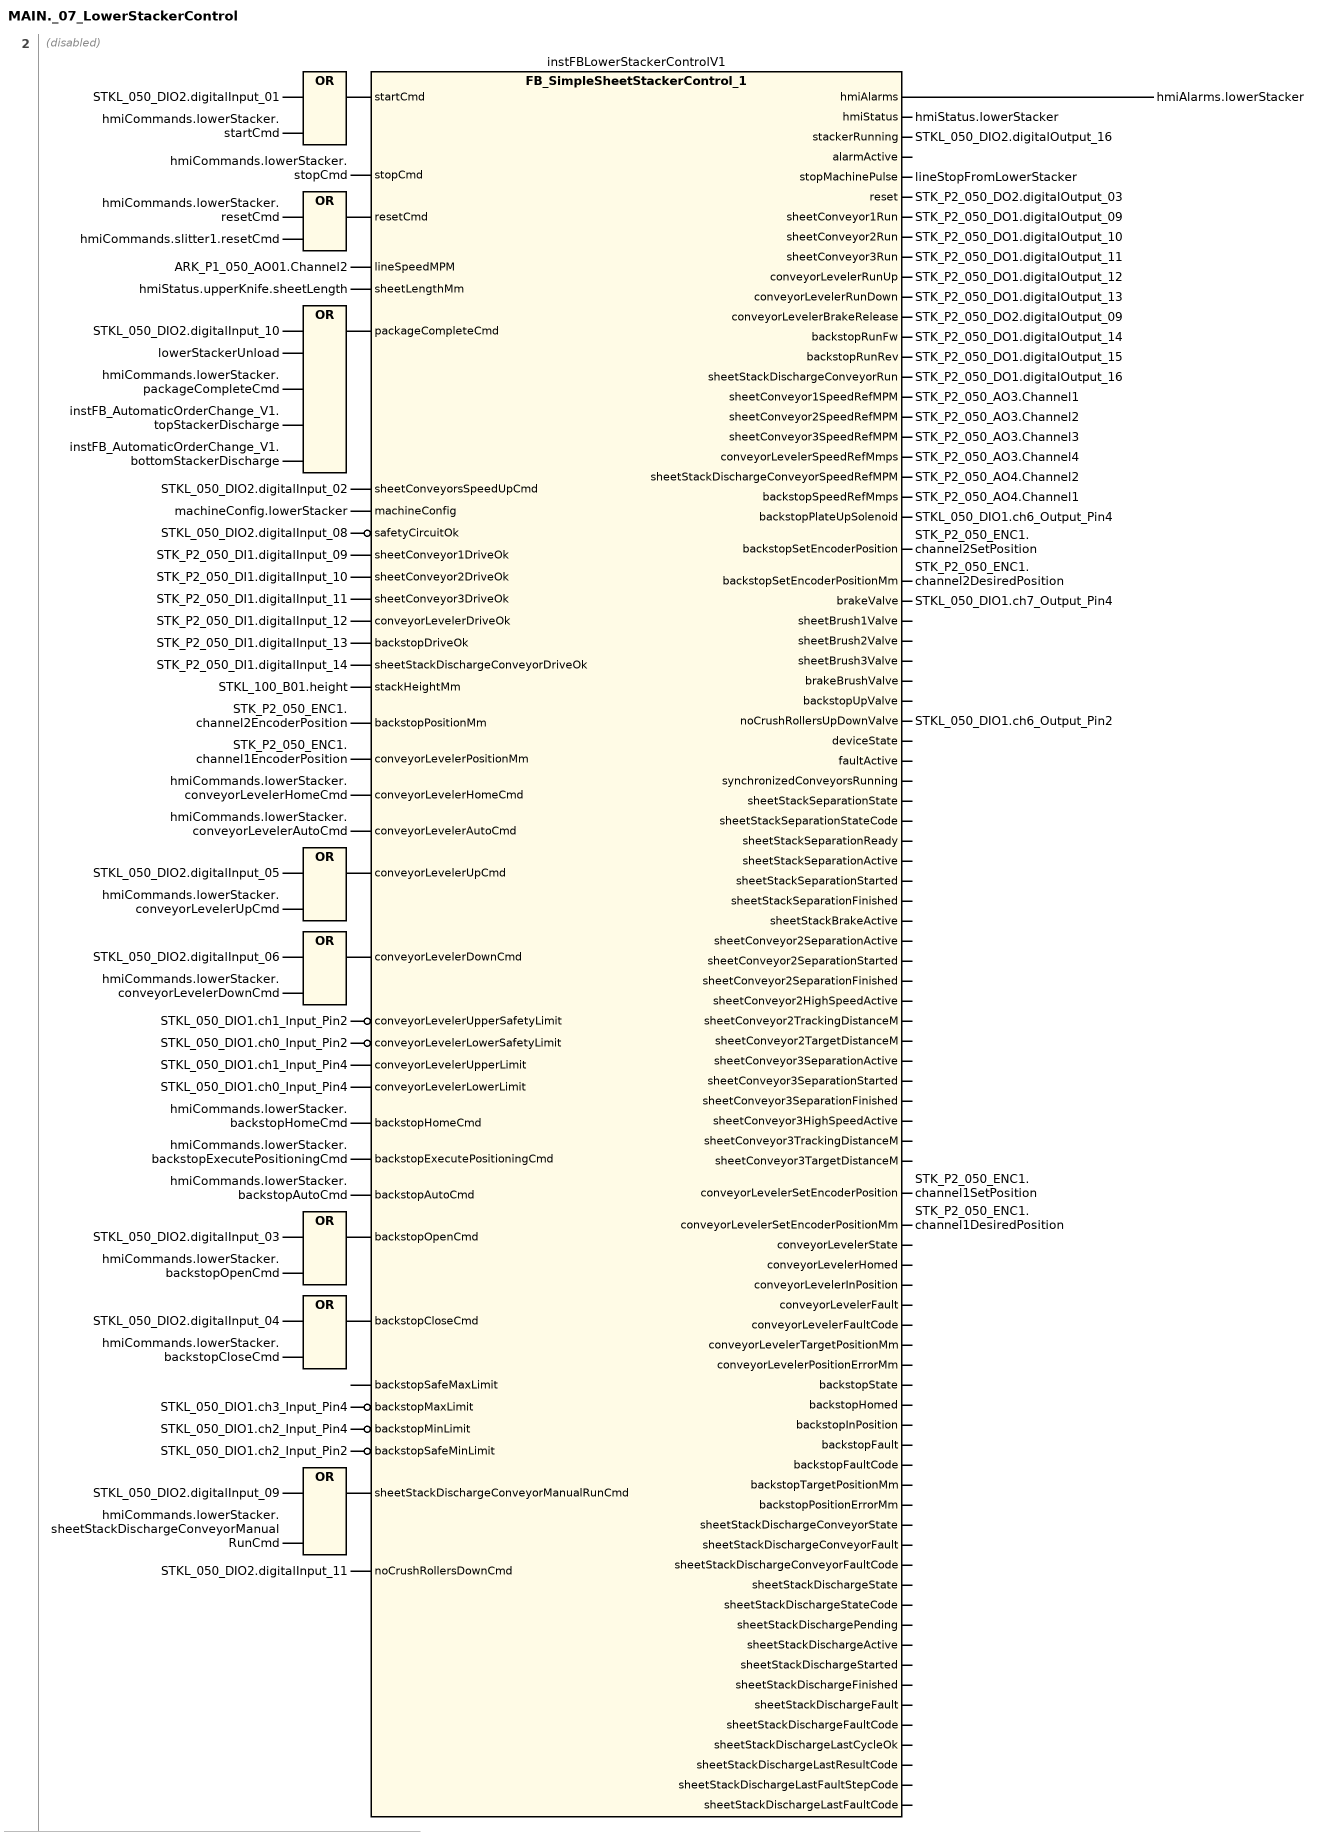
// NETWORK 2 (disabled)
// instFBLowerStackerControlV1(
//     startCmd := STKL_050_DIO2.digitalInput_01 OR hmiCommands.lowerStacker.startCmd,
//     stopCmd := hmiCommands.lowerStacker.stopCmd,
//     resetCmd := hmiCommands.lowerStacker.resetCmd OR hmiCommands.slitter1.resetCmd,
//     lineSpeedMPM := ARK_P1_050_AO01.Channel2,
//     sheetLengthMm := hmiStatus.upperKnife.sheetLength,
//     packageCompleteCmd := STKL_050_DIO2.digitalInput_10 OR lowerStackerUnload OR hmiCommands.lowerStacker.packageCompleteCmd OR instFB_AutomaticOrderChange_V1.topStackerDischarge OR instFB_AutomaticOrderChange_V1.bottomStackerDischarge,
//     sheetConveyorsSpeedUpCmd := STKL_050_DIO2.digitalInput_02,
//     machineConfig := machineConfig.lowerStacker,
//     safetyCircuitOk := NOT STKL_050_DIO2.digitalInput_08,
//     sheetConveyor1DriveOk := STK_P2_050_DI1.digitalInput_09,
//     sheetConveyor2DriveOk := STK_P2_050_DI1.digitalInput_10,
//     sheetConveyor3DriveOk := STK_P2_050_DI1.digitalInput_11,
//     conveyorLevelerDriveOk := STK_P2_050_DI1.digitalInput_12,
//     backstopDriveOk := STK_P2_050_DI1.digitalInput_13,
//     sheetStackDischargeConveyorDriveOk := STK_P2_050_DI1.digitalInput_14,
//     stackHeightMm := STKL_100_B01.height,
//     backstopPositionMm := STK_P2_050_ENC1.channel2EncoderPosition,
//     conveyorLevelerPositionMm := STK_P2_050_ENC1.channel1EncoderPosition,
//     conveyorLevelerHomeCmd := hmiCommands.lowerStacker.conveyorLevelerHomeCmd,
//     conveyorLevelerAutoCmd := hmiCommands.lowerStacker.conveyorLevelerAutoCmd,
//     conveyorLevelerUpCmd := STKL_050_DIO2.digitalInput_05 OR hmiCommands.lowerStacker.conveyorLevelerUpCmd,
//     conveyorLevelerDownCmd := STKL_050_DIO2.digitalInput_06 OR hmiCommands.lowerStacker.conveyorLevelerDownCmd,
//     conveyorLevelerUpperSafetyLimit := NOT STKL_050_DIO1.ch1_Input_Pin2,
//     conveyorLevelerLowerSafetyLimit := NOT STKL_050_DIO1.ch0_Input_Pin2,
//     conveyorLevelerUpperLimit := STKL_050_DIO1.ch1_Input_Pin4,
//     conveyorLevelerLowerLimit := STKL_050_DIO1.ch0_Input_Pin4,
//     backstopHomeCmd := hmiCommands.lowerStacker.backstopHomeCmd,
//     backstopExecutePositioningCmd := hmiCommands.lowerStacker.backstopExecutePositioningCmd,
//     backstopAutoCmd := hmiCommands.lowerStacker.backstopAutoCmd,
//     backstopOpenCmd := STKL_050_DIO2.digitalInput_03 OR hmiCommands.lowerStacker.backstopOpenCmd,
//     backstopCloseCmd := STKL_050_DIO2.digitalInput_04 OR hmiCommands.lowerStacker.backstopCloseCmd,
//     backstopMaxLimit := NOT STKL_050_DIO1.ch3_Input_Pin4,
//     backstopMinLimit := NOT STKL_050_DIO1.ch2_Input_Pin4,
//     backstopSafeMinLimit := NOT STKL_050_DIO1.ch2_Input_Pin2,
//     sheetStackDischargeConveyorManualRunCmd := STKL_050_DIO2.digitalInput_09 OR hmiCommands.lowerStacker.sheetStackDischargeConveyorManualRunCmd,
//     noCrushRollersDownCmd := STKL_050_DIO2.digitalInput_11,
//     hmiStatus => hmiStatus.lowerStacker,
//     stackerRunning => STKL_050_DIO2.digitalOutput_16,
//     stopMachinePulse => lineStopFromLowerStacker,
//     reset => STK_P2_050_DO2.digitalOutput_03,
//     sheetConveyor1Run => STK_P2_050_DO1.digitalOutput_09,
//     sheetConveyor2Run => STK_P2_050_DO1.digitalOutput_10,
//     sheetConveyor3Run => STK_P2_050_DO1.digitalOutput_11,
//     conveyorLevelerRunUp => STK_P2_050_DO1.digitalOutput_12,
//     conveyorLevelerRunDown => STK_P2_050_DO1.digitalOutput_13,
//     conveyorLevelerBrakeRelease => STK_P2_050_DO2.digitalOutput_09,
//     backstopRunFw => STK_P2_050_DO1.digitalOutput_14,
//     backstopRunRev => STK_P2_050_DO1.digitalOutput_15,
//     sheetStackDischargeConveyorRun => STK_P2_050_DO1.digitalOutput_16,
//     sheetConveyor1SpeedRefMPM => STK_P2_050_AO3.Channel1,
//     sheetConveyor2SpeedRefMPM => STK_P2_050_AO3.Channel2,
//     sheetConveyor3SpeedRefMPM => STK_P2_050_AO3.Channel3,
//     conveyorLevelerSpeedRefMmps => STK_P2_050_AO3.Channel4,
//     sheetStackDischargeConveyorSpeedRefMPM => STK_P2_050_AO4.Channel2,
//     backstopSpeedRefMmps => STK_P2_050_AO4.Channel1,
//     backstopPlateUpSolenoid => STKL_050_DIO1.ch6_Output_Pin4,
//     backstopSetEncoderPosition => STK_P2_050_ENC1.channel2SetPosition,
//     backstopSetEncoderPositionMm => STK_P2_050_ENC1.channel2DesiredPosition,
//     brakeValve => STKL_050_DIO1.ch7_Output_Pin4,
//     noCrushRollersUpDownValve => STKL_050_DIO1.ch6_Output_Pin2,
//     conveyorLevelerSetEncoderPosition => STK_P2_050_ENC1.channel1SetPosition,
//     conveyorLevelerSetEncoderPositionMm => STK_P2_050_ENC1.channel1DesiredPosition); // FB_SimpleSheetStackerControl_1
// hmiAlarms.lowerStacker := instFBLowerStackerControlV1.hmiAlarms;
END_METHOD

METHOD _08_UpperStackerControl
VAR_INPUT
END_VAR
//STKU_050_DIO2.digitalInput_12 Material no backstop
VAR

END_VAR
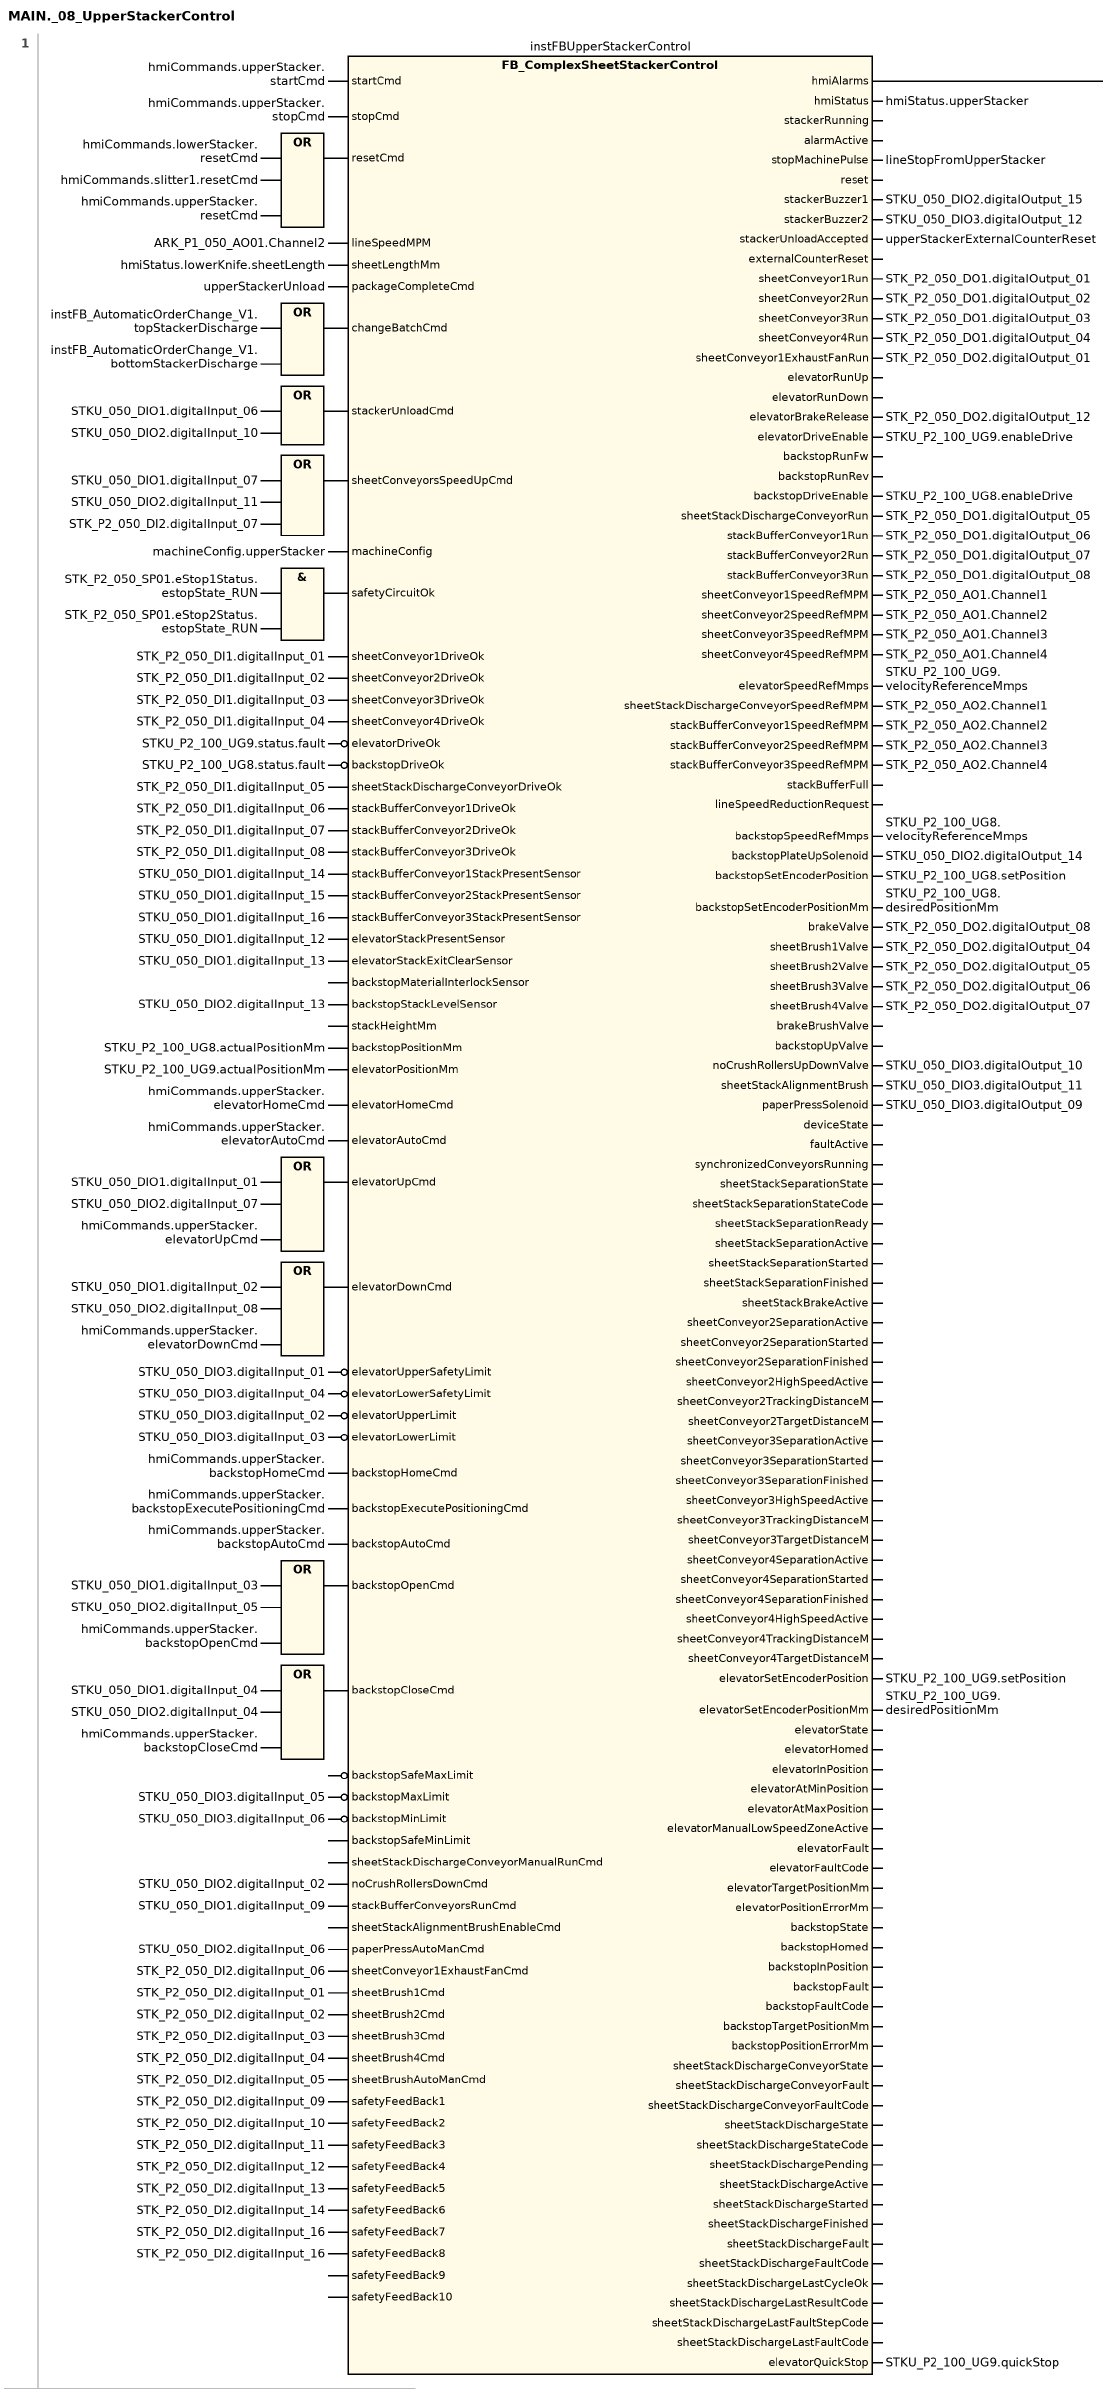
// NETWORK 1
instFBUpperStackerControl(
    startCmd := hmiCommands.upperStacker.startCmd,
    stopCmd := hmiCommands.upperStacker.stopCmd,
    resetCmd := hmiCommands.lowerStacker.resetCmd OR hmiCommands.slitter1.resetCmd OR hmiCommands.upperStacker.resetCmd,
    lineSpeedMPM := ARK_P1_050_AO01.Channel2,
    sheetLengthMm := hmiStatus.lowerKnife.sheetLength,
    packageCompleteCmd := upperStackerUnload,
    changeBatchCmd := instFB_AutomaticOrderChange_V1.topStackerDischarge OR instFB_AutomaticOrderChange_V1.bottomStackerDischarge,
    stackerUnloadCmd := STKU_050_DIO1.digitalInput_06 OR STKU_050_DIO2.digitalInput_10,
    sheetConveyorsSpeedUpCmd := STKU_050_DIO1.digitalInput_07 OR STKU_050_DIO2.digitalInput_11 OR STK_P2_050_DI2.digitalInput_07,
    machineConfig := machineConfig.upperStacker,
    safetyCircuitOk := STK_P2_050_SP01.eStop1Status.estopState_RUN AND STK_P2_050_SP01.eStop2Status.estopState_RUN,
    sheetConveyor1DriveOk := STK_P2_050_DI1.digitalInput_01,
    sheetConveyor2DriveOk := STK_P2_050_DI1.digitalInput_02,
    sheetConveyor3DriveOk := STK_P2_050_DI1.digitalInput_03,
    sheetConveyor4DriveOk := STK_P2_050_DI1.digitalInput_04,
    elevatorDriveOk := NOT STKU_P2_100_UG9.status.fault,
    backstopDriveOk := NOT STKU_P2_100_UG8.status.fault,
    sheetStackDischargeConveyorDriveOk := STK_P2_050_DI1.digitalInput_05,
    stackBufferConveyor1DriveOk := STK_P2_050_DI1.digitalInput_06,
    stackBufferConveyor2DriveOk := STK_P2_050_DI1.digitalInput_07,
    stackBufferConveyor3DriveOk := STK_P2_050_DI1.digitalInput_08,
    stackBufferConveyor1StackPresentSensor := STKU_050_DIO1.digitalInput_14,
    stackBufferConveyor2StackPresentSensor := STKU_050_DIO1.digitalInput_15,
    stackBufferConveyor3StackPresentSensor := STKU_050_DIO1.digitalInput_16,
    elevatorStackPresentSensor := STKU_050_DIO1.digitalInput_12,
    elevatorStackExitClearSensor := STKU_050_DIO1.digitalInput_13,
    backstopStackLevelSensor := STKU_050_DIO2.digitalInput_13,
    backstopPositionMm := STKU_P2_100_UG8.actualPositionMm,
    elevatorPositionMm := STKU_P2_100_UG9.actualPositionMm,
    elevatorHomeCmd := hmiCommands.upperStacker.elevatorHomeCmd,
    elevatorAutoCmd := hmiCommands.upperStacker.elevatorAutoCmd,
    elevatorUpCmd := STKU_050_DIO1.digitalInput_01 OR STKU_050_DIO2.digitalInput_07 OR hmiCommands.upperStacker.elevatorUpCmd,
    elevatorDownCmd := STKU_050_DIO1.digitalInput_02 OR STKU_050_DIO2.digitalInput_08 OR hmiCommands.upperStacker.elevatorDownCmd,
    elevatorUpperSafetyLimit := NOT STKU_050_DIO3.digitalInput_01,
    elevatorLowerSafetyLimit := NOT STKU_050_DIO3.digitalInput_04,
    elevatorUpperLimit := NOT STKU_050_DIO3.digitalInput_02,
    elevatorLowerLimit := NOT STKU_050_DIO3.digitalInput_03,
    backstopHomeCmd := hmiCommands.upperStacker.backstopHomeCmd,
    backstopExecutePositioningCmd := hmiCommands.upperStacker.backstopExecutePositioningCmd,
    backstopAutoCmd := hmiCommands.upperStacker.backstopAutoCmd,
    backstopOpenCmd := STKU_050_DIO1.digitalInput_03 OR STKU_050_DIO2.digitalInput_05 OR hmiCommands.upperStacker.backstopOpenCmd,
    backstopCloseCmd := STKU_050_DIO1.digitalInput_04 OR STKU_050_DIO2.digitalInput_04 OR hmiCommands.upperStacker.backstopCloseCmd,
    backstopMaxLimit := NOT STKU_050_DIO3.digitalInput_05,
    backstopMinLimit := NOT STKU_050_DIO3.digitalInput_06,
    noCrushRollersDownCmd := STKU_050_DIO2.digitalInput_02,
    stackBufferConveyorsRunCmd := STKU_050_DIO1.digitalInput_09,
    paperPressAutoManCmd := STKU_050_DIO2.digitalInput_06,
    sheetConveyor1ExhaustFanCmd := STK_P2_050_DI2.digitalInput_06,
    sheetBrush1Cmd := STK_P2_050_DI2.digitalInput_01,
    sheetBrush2Cmd := STK_P2_050_DI2.digitalInput_02,
    sheetBrush3Cmd := STK_P2_050_DI2.digitalInput_03,
    sheetBrush4Cmd := STK_P2_050_DI2.digitalInput_04,
    sheetBrushAutoManCmd := STK_P2_050_DI2.digitalInput_05,
    safetyFeedBack1 := STK_P2_050_DI2.digitalInput_09,
    safetyFeedBack2 := STK_P2_050_DI2.digitalInput_10,
    safetyFeedBack3 := STK_P2_050_DI2.digitalInput_11,
    safetyFeedBack4 := STK_P2_050_DI2.digitalInput_12,
    safetyFeedBack5 := STK_P2_050_DI2.digitalInput_13,
    safetyFeedBack6 := STK_P2_050_DI2.digitalInput_14,
    safetyFeedBack7 := STK_P2_050_DI2.digitalInput_16,
    safetyFeedBack8 := STK_P2_050_DI2.digitalInput_16,
    hmiStatus => hmiStatus.upperStacker,
    stopMachinePulse => lineStopFromUpperStacker,
    stackerBuzzer1 => STKU_050_DIO2.digitalOutput_15,
    stackerBuzzer2 => STKU_050_DIO3.digitalOutput_12,
    stackerUnloadAccepted => upperStackerExternalCounterReset,
    sheetConveyor1Run => STK_P2_050_DO1.digitalOutput_01,
    sheetConveyor2Run => STK_P2_050_DO1.digitalOutput_02,
    sheetConveyor3Run => STK_P2_050_DO1.digitalOutput_03,
    sheetConveyor4Run => STK_P2_050_DO1.digitalOutput_04,
    sheetConveyor1ExhaustFanRun => STK_P2_050_DO2.digitalOutput_01,
    elevatorBrakeRelease => STK_P2_050_DO2.digitalOutput_12,
    elevatorDriveEnable => STKU_P2_100_UG9.enableDrive,
    backstopDriveEnable => STKU_P2_100_UG8.enableDrive,
    sheetStackDischargeConveyorRun => STK_P2_050_DO1.digitalOutput_05,
    stackBufferConveyor1Run => STK_P2_050_DO1.digitalOutput_06,
    stackBufferConveyor2Run => STK_P2_050_DO1.digitalOutput_07,
    stackBufferConveyor3Run => STK_P2_050_DO1.digitalOutput_08,
    sheetConveyor1SpeedRefMPM => STK_P2_050_AO1.Channel1,
    sheetConveyor2SpeedRefMPM => STK_P2_050_AO1.Channel2,
    sheetConveyor3SpeedRefMPM => STK_P2_050_AO1.Channel3,
    sheetConveyor4SpeedRefMPM => STK_P2_050_AO1.Channel4,
    elevatorSpeedRefMmps => STKU_P2_100_UG9.velocityReferenceMmps,
    sheetStackDischargeConveyorSpeedRefMPM => STK_P2_050_AO2.Channel1,
    stackBufferConveyor1SpeedRefMPM => STK_P2_050_AO2.Channel2,
    stackBufferConveyor2SpeedRefMPM => STK_P2_050_AO2.Channel3,
    stackBufferConveyor3SpeedRefMPM => STK_P2_050_AO2.Channel4,
    backstopSpeedRefMmps => STKU_P2_100_UG8.velocityReferenceMmps,
    backstopPlateUpSolenoid => STKU_050_DIO2.digitalOutput_14,
    backstopSetEncoderPosition => STKU_P2_100_UG8.setPosition,
    backstopSetEncoderPositionMm => STKU_P2_100_UG8.desiredPositionMm,
    brakeValve => STK_P2_050_DO2.digitalOutput_08,
    sheetBrush1Valve => STK_P2_050_DO2.digitalOutput_04,
    sheetBrush2Valve => STK_P2_050_DO2.digitalOutput_05,
    sheetBrush3Valve => STK_P2_050_DO2.digitalOutput_06,
    sheetBrush4Valve => STK_P2_050_DO2.digitalOutput_07,
    noCrushRollersUpDownValve => STKU_050_DIO3.digitalOutput_10,
    sheetStackAlignmentBrush => STKU_050_DIO3.digitalOutput_11,
    paperPressSolenoid => STKU_050_DIO3.digitalOutput_09,
    elevatorSetEncoderPosition => STKU_P2_100_UG9.setPosition,
    elevatorSetEncoderPositionMm => STKU_P2_100_UG9.desiredPositionMm,
    elevatorQuickStop => STKU_P2_100_UG9.quickStop); // FB_ComplexSheetStackerControl
END_METHOD

ACTION ACT_Slitter1Control:
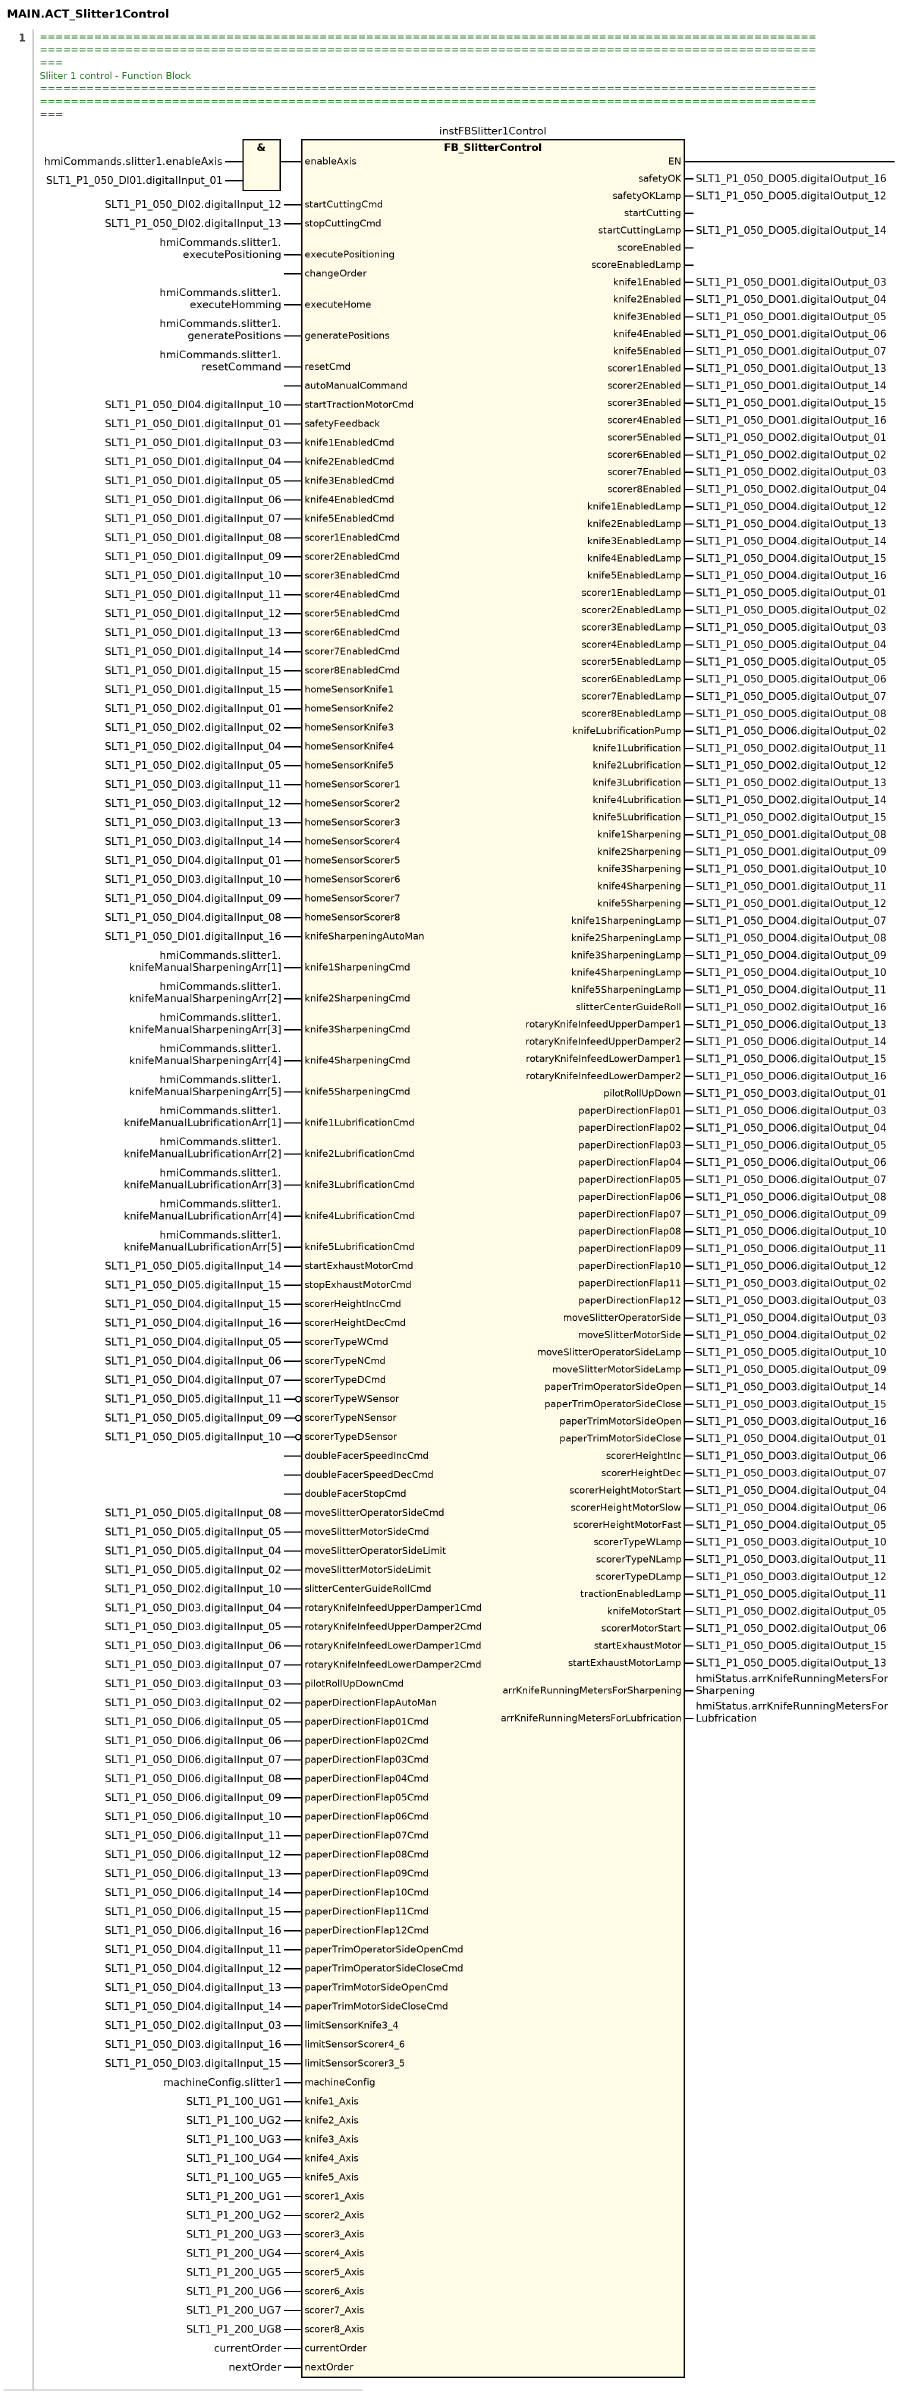
// NETWORK 1
// 					===========================================================================================================================================================================================================
//
// Sliiter 1 control - Function Block
//
// ===========================================================================================================================================================================================================
//
instFBSlitter1Control(
    enableAxis := hmiCommands.slitter1.enableAxis AND SLT1_P1_050_DI01.digitalInput_01,
    startCuttingCmd := SLT1_P1_050_DI02.digitalInput_12,
    stopCuttingCmd := SLT1_P1_050_DI02.digitalInput_13,
    executePositioning := hmiCommands.slitter1.executePositioning,
    executeHome := hmiCommands.slitter1.executeHomming,
    generatePositions := hmiCommands.slitter1.generatePositions,
    resetCmd := hmiCommands.slitter1.resetCommand,
    startTractionMotorCmd := SLT1_P1_050_DI04.digitalInput_10,
    safetyFeedback := SLT1_P1_050_DI01.digitalInput_01,
    knife1EnabledCmd := SLT1_P1_050_DI01.digitalInput_03,
    knife2EnabledCmd := SLT1_P1_050_DI01.digitalInput_04,
    knife3EnabledCmd := SLT1_P1_050_DI01.digitalInput_05,
    knife4EnabledCmd := SLT1_P1_050_DI01.digitalInput_06,
    knife5EnabledCmd := SLT1_P1_050_DI01.digitalInput_07,
    scorer1EnabledCmd := SLT1_P1_050_DI01.digitalInput_08,
    scorer2EnabledCmd := SLT1_P1_050_DI01.digitalInput_09,
    scorer3EnabledCmd := SLT1_P1_050_DI01.digitalInput_10,
    scorer4EnabledCmd := SLT1_P1_050_DI01.digitalInput_11,
    scorer5EnabledCmd := SLT1_P1_050_DI01.digitalInput_12,
    scorer6EnabledCmd := SLT1_P1_050_DI01.digitalInput_13,
    scorer7EnabledCmd := SLT1_P1_050_DI01.digitalInput_14,
    scorer8EnabledCmd := SLT1_P1_050_DI01.digitalInput_15,
    homeSensorKnife1 := SLT1_P1_050_DI01.digitalInput_15,
    homeSensorKnife2 := SLT1_P1_050_DI02.digitalInput_01,
    homeSensorKnife3 := SLT1_P1_050_DI02.digitalInput_02,
    homeSensorKnife4 := SLT1_P1_050_DI02.digitalInput_04,
    homeSensorKnife5 := SLT1_P1_050_DI02.digitalInput_05,
    homeSensorScorer1 := SLT1_P1_050_DI03.digitalInput_11,
    homeSensorScorer2 := SLT1_P1_050_DI03.digitalInput_12,
    homeSensorScorer3 := SLT1_P1_050_DI03.digitalInput_13,
    homeSensorScorer4 := SLT1_P1_050_DI03.digitalInput_14,
    homeSensorScorer5 := SLT1_P1_050_DI04.digitalInput_01,
    homeSensorScorer6 := SLT1_P1_050_DI03.digitalInput_10,
    homeSensorScorer7 := SLT1_P1_050_DI04.digitalInput_09,
    homeSensorScorer8 := SLT1_P1_050_DI04.digitalInput_08,
    knifeSharpeningAutoMan := SLT1_P1_050_DI01.digitalInput_16,
    knife1SharpeningCmd := hmiCommands.slitter1.knifeManualSharpeningArr[1],
    knife2SharpeningCmd := hmiCommands.slitter1.knifeManualSharpeningArr[2],
    knife3SharpeningCmd := hmiCommands.slitter1.knifeManualSharpeningArr[3],
    knife4SharpeningCmd := hmiCommands.slitter1.knifeManualSharpeningArr[4],
    knife5SharpeningCmd := hmiCommands.slitter1.knifeManualSharpeningArr[5],
    knife1LubrificationCmd := hmiCommands.slitter1.knifeManualLubrificationArr[1],
    knife2LubrificationCmd := hmiCommands.slitter1.knifeManualLubrificationArr[2],
    knife3LubrificationCmd := hmiCommands.slitter1.knifeManualLubrificationArr[3],
    knife4LubrificationCmd := hmiCommands.slitter1.knifeManualLubrificationArr[4],
    knife5LubrificationCmd := hmiCommands.slitter1.knifeManualLubrificationArr[5],
    startExhaustMotorCmd := SLT1_P1_050_DI05.digitalInput_14,
    stopExhaustMotorCmd := SLT1_P1_050_DI05.digitalInput_15,
    scorerHeightIncCmd := SLT1_P1_050_DI04.digitalInput_15,
    scorerHeightDecCmd := SLT1_P1_050_DI04.digitalInput_16,
    scorerTypeWCmd := SLT1_P1_050_DI04.digitalInput_05,
    scorerTypeNCmd := SLT1_P1_050_DI04.digitalInput_06,
    scorerTypeDCmd := SLT1_P1_050_DI04.digitalInput_07,
    scorerTypeWSensor := NOT SLT1_P1_050_DI05.digitalInput_11,
    scorerTypeNSensor := NOT SLT1_P1_050_DI05.digitalInput_09,
    scorerTypeDSensor := NOT SLT1_P1_050_DI05.digitalInput_10,
    moveSlitterOperatorSideCmd := SLT1_P1_050_DI05.digitalInput_08,
    moveSlitterMotorSideCmd := SLT1_P1_050_DI05.digitalInput_05,
    moveSlitterOperatorSideLimit := SLT1_P1_050_DI05.digitalInput_04,
    moveSlitterMotorSideLimit := SLT1_P1_050_DI05.digitalInput_02,
    slitterCenterGuideRollCmd := SLT1_P1_050_DI02.digitalInput_10,
    rotaryKnifeInfeedUpperDamper1Cmd := SLT1_P1_050_DI03.digitalInput_04,
    rotaryKnifeInfeedUpperDamper2Cmd := SLT1_P1_050_DI03.digitalInput_05,
    rotaryKnifeInfeedLowerDamper1Cmd := SLT1_P1_050_DI03.digitalInput_06,
    rotaryKnifeInfeedLowerDamper2Cmd := SLT1_P1_050_DI03.digitalInput_07,
    pilotRollUpDownCmd := SLT1_P1_050_DI03.digitalInput_03,
    paperDirectionFlapAutoMan := SLT1_P1_050_DI03.digitalInput_02,
    paperDirectionFlap01Cmd := SLT1_P1_050_DI06.digitalInput_05,
    paperDirectionFlap02Cmd := SLT1_P1_050_DI06.digitalInput_06,
    paperDirectionFlap03Cmd := SLT1_P1_050_DI06.digitalInput_07,
    paperDirectionFlap04Cmd := SLT1_P1_050_DI06.digitalInput_08,
    paperDirectionFlap05Cmd := SLT1_P1_050_DI06.digitalInput_09,
    paperDirectionFlap06Cmd := SLT1_P1_050_DI06.digitalInput_10,
    paperDirectionFlap07Cmd := SLT1_P1_050_DI06.digitalInput_11,
    paperDirectionFlap08Cmd := SLT1_P1_050_DI06.digitalInput_12,
    paperDirectionFlap09Cmd := SLT1_P1_050_DI06.digitalInput_13,
    paperDirectionFlap10Cmd := SLT1_P1_050_DI06.digitalInput_14,
    paperDirectionFlap11Cmd := SLT1_P1_050_DI06.digitalInput_15,
    paperDirectionFlap12Cmd := SLT1_P1_050_DI06.digitalInput_16,
    paperTrimOperatorSideOpenCmd := SLT1_P1_050_DI04.digitalInput_11,
    paperTrimOperatorSideCloseCmd := SLT1_P1_050_DI04.digitalInput_12,
    paperTrimMotorSideOpenCmd := SLT1_P1_050_DI04.digitalInput_13,
    paperTrimMotorSideCloseCmd := SLT1_P1_050_DI04.digitalInput_14,
    limitSensorKnife3_4 := SLT1_P1_050_DI02.digitalInput_03,
    limitSensorScorer4_6 := SLT1_P1_050_DI03.digitalInput_16,
    limitSensorScorer3_5 := SLT1_P1_050_DI03.digitalInput_15,
    machineConfig := machineConfig.slitter1,
    knife1_Axis := SLT1_P1_100_UG1,
    knife2_Axis := SLT1_P1_100_UG2,
    knife3_Axis := SLT1_P1_100_UG3,
    knife4_Axis := SLT1_P1_100_UG4,
    knife5_Axis := SLT1_P1_100_UG5,
    scorer1_Axis := SLT1_P1_200_UG1,
    scorer2_Axis := SLT1_P1_200_UG2,
    scorer3_Axis := SLT1_P1_200_UG3,
    scorer4_Axis := SLT1_P1_200_UG4,
    scorer5_Axis := SLT1_P1_200_UG5,
    scorer6_Axis := SLT1_P1_200_UG6,
    scorer7_Axis := SLT1_P1_200_UG7,
    scorer8_Axis := SLT1_P1_200_UG8,
    currentOrder := currentOrder,
    nextOrder := nextOrder,
    safetyOK => SLT1_P1_050_DO05.digitalOutput_16,
    safetyOKLamp => SLT1_P1_050_DO05.digitalOutput_12,
    startCuttingLamp => SLT1_P1_050_DO05.digitalOutput_14,
    knife1Enabled => SLT1_P1_050_DO01.digitalOutput_03,
    knife2Enabled => SLT1_P1_050_DO01.digitalOutput_04,
    knife3Enabled => SLT1_P1_050_DO01.digitalOutput_05,
    knife4Enabled => SLT1_P1_050_DO01.digitalOutput_06,
    knife5Enabled => SLT1_P1_050_DO01.digitalOutput_07,
    scorer1Enabled => SLT1_P1_050_DO01.digitalOutput_13,
    scorer2Enabled => SLT1_P1_050_DO01.digitalOutput_14,
    scorer3Enabled => SLT1_P1_050_DO01.digitalOutput_15,
    scorer4Enabled => SLT1_P1_050_DO01.digitalOutput_16,
    scorer5Enabled => SLT1_P1_050_DO02.digitalOutput_01,
    scorer6Enabled => SLT1_P1_050_DO02.digitalOutput_02,
    scorer7Enabled => SLT1_P1_050_DO02.digitalOutput_03,
    scorer8Enabled => SLT1_P1_050_DO02.digitalOutput_04,
    knife1EnabledLamp => SLT1_P1_050_DO04.digitalOutput_12,
    knife2EnabledLamp => SLT1_P1_050_DO04.digitalOutput_13,
    knife3EnabledLamp => SLT1_P1_050_DO04.digitalOutput_14,
    knife4EnabledLamp => SLT1_P1_050_DO04.digitalOutput_15,
    knife5EnabledLamp => SLT1_P1_050_DO04.digitalOutput_16,
    scorer1EnabledLamp => SLT1_P1_050_DO05.digitalOutput_01,
    scorer2EnabledLamp => SLT1_P1_050_DO05.digitalOutput_02,
    scorer3EnabledLamp => SLT1_P1_050_DO05.digitalOutput_03,
    scorer4EnabledLamp => SLT1_P1_050_DO05.digitalOutput_04,
    scorer5EnabledLamp => SLT1_P1_050_DO05.digitalOutput_05,
    scorer6EnabledLamp => SLT1_P1_050_DO05.digitalOutput_06,
    scorer7EnabledLamp => SLT1_P1_050_DO05.digitalOutput_07,
    scorer8EnabledLamp => SLT1_P1_050_DO05.digitalOutput_08,
    knifeLubrificationPump => SLT1_P1_050_DO06.digitalOutput_02,
    knife1Lubrification => SLT1_P1_050_DO02.digitalOutput_11,
    knife2Lubrification => SLT1_P1_050_DO02.digitalOutput_12,
    knife3Lubrification => SLT1_P1_050_DO02.digitalOutput_13,
    knife4Lubrification => SLT1_P1_050_DO02.digitalOutput_14,
    knife5Lubrification => SLT1_P1_050_DO02.digitalOutput_15,
    knife1Sharpening => SLT1_P1_050_DO01.digitalOutput_08,
    knife2Sharpening => SLT1_P1_050_DO01.digitalOutput_09,
    knife3Sharpening => SLT1_P1_050_DO01.digitalOutput_10,
    knife4Sharpening => SLT1_P1_050_DO01.digitalOutput_11,
    knife5Sharpening => SLT1_P1_050_DO01.digitalOutput_12,
    knife1SharpeningLamp => SLT1_P1_050_DO04.digitalOutput_07,
    knife2SharpeningLamp => SLT1_P1_050_DO04.digitalOutput_08,
    knife3SharpeningLamp => SLT1_P1_050_DO04.digitalOutput_09,
    knife4SharpeningLamp => SLT1_P1_050_DO04.digitalOutput_10,
    knife5SharpeningLamp => SLT1_P1_050_DO04.digitalOutput_11,
    slitterCenterGuideRoll => SLT1_P1_050_DO02.digitalOutput_16,
    rotaryKnifeInfeedUpperDamper1 => SLT1_P1_050_DO06.digitalOutput_13,
    rotaryKnifeInfeedUpperDamper2 => SLT1_P1_050_DO06.digitalOutput_14,
    rotaryKnifeInfeedLowerDamper1 => SLT1_P1_050_DO06.digitalOutput_15,
    rotaryKnifeInfeedLowerDamper2 => SLT1_P1_050_DO06.digitalOutput_16,
    pilotRollUpDown => SLT1_P1_050_DO03.digitalOutput_01,
    paperDirectionFlap01 => SLT1_P1_050_DO06.digitalOutput_03,
    paperDirectionFlap02 => SLT1_P1_050_DO06.digitalOutput_04,
    paperDirectionFlap03 => SLT1_P1_050_DO06.digitalOutput_05,
    paperDirectionFlap04 => SLT1_P1_050_DO06.digitalOutput_06,
    paperDirectionFlap05 => SLT1_P1_050_DO06.digitalOutput_07,
    paperDirectionFlap06 => SLT1_P1_050_DO06.digitalOutput_08,
    paperDirectionFlap07 => SLT1_P1_050_DO06.digitalOutput_09,
    paperDirectionFlap08 => SLT1_P1_050_DO06.digitalOutput_10,
    paperDirectionFlap09 => SLT1_P1_050_DO06.digitalOutput_11,
    paperDirectionFlap10 => SLT1_P1_050_DO06.digitalOutput_12,
    paperDirectionFlap11 => SLT1_P1_050_DO03.digitalOutput_02,
    paperDirectionFlap12 => SLT1_P1_050_DO03.digitalOutput_03,
    moveSlitterOperatorSide => SLT1_P1_050_DO04.digitalOutput_03,
    moveSlitterMotorSide => SLT1_P1_050_DO04.digitalOutput_02,
    moveSlitterOperatorSideLamp => SLT1_P1_050_DO05.digitalOutput_10,
    moveSlitterMotorSideLamp => SLT1_P1_050_DO05.digitalOutput_09,
    paperTrimOperatorSideOpen => SLT1_P1_050_DO03.digitalOutput_14,
    paperTrimOperatorSideClose => SLT1_P1_050_DO03.digitalOutput_15,
    paperTrimMotorSideOpen => SLT1_P1_050_DO03.digitalOutput_16,
    paperTrimMotorSideClose => SLT1_P1_050_DO04.digitalOutput_01,
    scorerHeightInc => SLT1_P1_050_DO03.digitalOutput_06,
    scorerHeightDec => SLT1_P1_050_DO03.digitalOutput_07,
    scorerHeightMotorStart => SLT1_P1_050_DO04.digitalOutput_04,
    scorerHeightMotorSlow => SLT1_P1_050_DO04.digitalOutput_06,
    scorerHeightMotorFast => SLT1_P1_050_DO04.digitalOutput_05,
    scorerTypeWLamp => SLT1_P1_050_DO03.digitalOutput_10,
    scorerTypeNLamp => SLT1_P1_050_DO03.digitalOutput_11,
    scorerTypeDLamp => SLT1_P1_050_DO03.digitalOutput_12,
    tractionEnabledLamp => SLT1_P1_050_DO05.digitalOutput_11,
    knifeMotorStart => SLT1_P1_050_DO02.digitalOutput_05,
    scorerMotorStart => SLT1_P1_050_DO02.digitalOutput_06,
    startExhaustMotor => SLT1_P1_050_DO05.digitalOutput_15,
    startExhaustMotorLamp => SLT1_P1_050_DO05.digitalOutput_13,
    arrKnifeRunningMetersForSharpening => hmiStatus.arrKnifeRunningMetersForSharpening,
    arrKnifeRunningMetersForLubfrication => hmiStatus.arrKnifeRunningMetersForLubfrication); // FB_SlitterControl
END_ACTION

END_PROGRAM

// ---- Library/Machine/Slitter/FunctionBlocks/FB_SlitterControl.TcPOU
FUNCTION_BLOCK FB_SlitterControl
VAR_INPUT
    // General control commands
    enableAxis              : BOOL;  // Enable/disable positioning axis motors
    startCuttingCmd            : BOOL;  // Start slitter cutting process\
    stopCuttingCmd            : BOOL;  // Stop slitter cutting process\
		
    executePositioning      : BOOL;  // Execute positioning sequence
    changeOrder             : BOOL;  // Execute Automatic Order Change (AOC)
    executeHome             : BOOL;  // Execute slitter homing
    generatePositions       : BOOL;  // Generate knife/scorer positions
    resetCmd                : BOOL;  // Reset commands and states
    autoManualCommand       : BOOL;  // Mode selection [FALSE = Auto / TRUE = Manual]
	
	startTractionMotorCmd	: BOOL;


	lineSpeedMPM			: REAL;
	aocSpeedMPM				: REAL;
	aocRunning				: BOOL;


    outfeedRoll_ManCmd      : BOOL; // Manual Mode activation command
    
    outfeedRoll_UpCmd       : BOOL; // Manual command to raise the roll
    outfeedRoll_DownCmd     : BOOL; // Manual command to lower the roll

	
	safetyFeedback			: BOOL;
	
	paperPresenceSensor				: BOOL;
	measuringWheelPaperPresenceSensor		: BOOL;
	rotaryShearCutPulse					: BOOL;	
	measuringWheelPulseSensor		: BOOL;	
	
	    // Knife solenoid enable outputs
    knife1EnabledCmd           : BOOL;
    knife2EnabledCmd           : BOOL;
    knife3EnabledCmd           : BOOL;
    knife4EnabledCmd           : BOOL;
    knife5EnabledCmd           : BOOL;

    // Scorer solenoid enable outputs
    scorer1EnabledCmd          : BOOL;
    scorer2EnabledCmd          : BOOL;
    scorer3EnabledCmd          : BOOL;
    scorer4EnabledCmd          : BOOL;
    scorer5EnabledCmd          : BOOL;
    scorer6EnabledCmd          : BOOL;
    scorer7EnabledCmd          : BOOL;
    scorer8EnabledCmd          : BOOL;

    // Knife home sensors
	
    homeSensorKnife1        : BOOL;
    homeSensorKnife2        : BOOL;
    homeSensorKnife3        : BOOL;
    homeSensorKnife4        : BOOL;
    homeSensorKnife5        : BOOL;
    
    // Scorer home sensors
    homeSensorScorer1       : BOOL;
    homeSensorScorer2       : BOOL;
    homeSensorScorer3       : BOOL;
    homeSensorScorer4       : BOOL;
    homeSensorScorer5       : BOOL;
    homeSensorScorer6       : BOOL;
    homeSensorScorer7       : BOOL;
    homeSensorScorer8       : BOOL;
	
    // Knife sharpening
	
	knifeSharpeningAutoMan		: BOOL;	//Knife sharpening (0 = Manual / 1 = Auto)
    knife1SharpeningCmd        : BOOL;
    knife2SharpeningCmd        : BOOL;
    knife3SharpeningCmd        : BOOL;
    knife4SharpeningCmd        : BOOL;
    knife5SharpeningCmd        : BOOL;	

    knife1LubrificationCmd        : BOOL;
    knife2LubrificationCmd        : BOOL;
    knife3LubrificationCmd        : BOOL;
    knife4LubrificationCmd        : BOOL;
    knife5LubrificationCmd        : BOOL;		

	startExhaustMotorCmd				: BOOL;
	stopExhaustMotorCmd				: BOOL;

	
	scorerHeightIncCmd		: BOOL;	
	scorerHeightDecCmd		: BOOL;	
	
	scorerTypeWCmd	: BOOL;
	scorerTypeNCmd	: BOOL;	
	scorerTypeDCmd	: BOOL;	
	
	scorerTypeWSensor	: BOOL;
	scorerTypeNSensor	: BOOL;	
	scorerTypeDSensor	: BOOL;	
	

	doubleFacerSpeedIncCmd			: BOOL;	
	doubleFacerSpeedDecCmd			: BOOL;	
	doubleFacerStopCmd			: BOOL;
	
    // Slitter movement controls
    moveSlitterOperatorSideCmd : BOOL;
    moveSlitterMotorSideCmd    : BOOL;
    moveSlitterOperatorSideLimit : BOOL;
    moveSlitterMotorSideLimit    : BOOL;	

	
	slitterCenterGuideRollCmd		: BOOL;
	
	rotaryKnifeInfeedUpperDamper1Cmd : BOOL;
	rotaryKnifeInfeedUpperDamper2Cmd : BOOL;
	
	rotaryKnifeInfeedLowerDamper1Cmd : BOOL;
	rotaryKnifeInfeedLowerDamper2Cmd : BOOL;
	
	pilotRollUpDownCmd			: BOOL;
	
	
    // Paper direction flaps
	
	paperDirectionFlapAutoMan	: BOOL; // Paper direction flap (0=Manual / 1=Auto)
    paperDirectionFlap01Cmd    : BOOL;
    paperDirectionFlap02Cmd    : BOOL;
    paperDirectionFlap03Cmd    : BOOL;
    paperDirectionFlap04Cmd    : BOOL;
    paperDirectionFlap05Cmd    : BOOL;
    paperDirectionFlap06Cmd    : BOOL;
    paperDirectionFlap07Cmd    : BOOL;
    paperDirectionFlap08Cmd    : BOOL;
    paperDirectionFlap09Cmd    : BOOL;
    paperDirectionFlap10Cmd    : BOOL;
    paperDirectionFlap11Cmd    : BOOL;
    paperDirectionFlap12Cmd    : BOOL;

	flapsManualCmdArr	: ARRAY [1..27] OF hmiCommandsFlaps_TypeStruct;
	
	
	    // Paper scrap controls
    paperTrimOperatorSideOpenCmd  : BOOL;
    paperTrimOperatorSideCloseCmd : BOOL;
    paperTrimMotorSideOpenCmd     : BOOL;
    paperTrimMotorSideCloseCmd    : BOOL;
	
    // Limit sensors
    limitSensorKnife3_4     : BOOL;  // Between knife 3 and knife 4
    limitSensorScorer4_6    : BOOL;  // Between scorer 4 and scorer 6
    limitSensorScorer3_5    : BOOL;  // Between scorer 3 and scorer 5
	
	
	knifeManualSharpeningCmdArr		: ARRAY [1..20] OF BOOL;	(*This array is used to sharpen the knife manualy*)
	knifeManualLubrificationCmdArr		: ARRAY [1..20] OF BOOL;	(*This array is used to lubrificate the knife manualy*)

    // Machine configuration
    machineConfig           : slitterConfig_TypeStruct;
END_VAR

VAR_IN_OUT
    // Knife axes references
    knife1_Axis             : AXIS_REF;
    knife2_Axis             : AXIS_REF;
    knife3_Axis             : AXIS_REF;
    knife4_Axis             : AXIS_REF;
    knife5_Axis             : AXIS_REF;

    // Scorer axes references
    scorer1_Axis            : AXIS_REF;
    scorer2_Axis            : AXIS_REF;
    scorer3_Axis            : AXIS_REF;
    scorer4_Axis            : AXIS_REF;
    scorer5_Axis            : AXIS_REF;
    scorer6_Axis            : AXIS_REF;
    scorer7_Axis            : AXIS_REF;
    scorer8_Axis            : AXIS_REF;
    
    // Orders
    currentOrder            : Order_TypeStruct;
    nextOrder               : Order_TypeStruct;
END_VAR

VAR_OUTPUT
    EN                      : BOOL;  // Function block enabled

	safetyOK				: BOOL;
	safetyOKLamp			: BOOL;
	
	startCutting            : BOOL;  // Start slitter cutting process\
	startCuttingLamp        : BOOL;  // Start slitter cutting process\
	
	scoreEnabled			: BOOL;
	scoreEnabledLamp		: BOOL;
    homeFinished                        : BOOL;



    // Knife solenoid enable outputs
    knife1Enabled           : BOOL;
    knife2Enabled           : BOOL;
    knife3Enabled           : BOOL;
    knife4Enabled           : BOOL;
    knife5Enabled           : BOOL;

    // Scorer solenoid enable outputs
    scorer1Enabled          : BOOL;
    scorer2Enabled          : BOOL;
    scorer3Enabled          : BOOL;
    scorer4Enabled          : BOOL;
    scorer5Enabled          : BOOL;
    scorer6Enabled          : BOOL;
    scorer7Enabled          : BOOL;
    scorer8Enabled          : BOOL;

    // Knife enabled indicator lamps
    knife1EnabledLamp       : BOOL;
    knife2EnabledLamp       : BOOL;
    knife3EnabledLamp       : BOOL;
    knife4EnabledLamp       : BOOL;
    knife5EnabledLamp       : BOOL;

    // Scorer enabled indicator lamps
    scorer1EnabledLamp      : BOOL;
    scorer2EnabledLamp      : BOOL;
    scorer3EnabledLamp      : BOOL;
    scorer4EnabledLamp      : BOOL;
    scorer5EnabledLamp      : BOOL;
    scorer6EnabledLamp      : BOOL;
    scorer7EnabledLamp      : BOOL;
    scorer8EnabledLamp      : BOOL;

    // Knife lubrication
    knifeLubrificationPump  : BOOL;  // Main lubrication pump
    knife1Lubrification     : BOOL;
    knife2Lubrification     : BOOL;
    knife3Lubrification     : BOOL;
    knife4Lubrification     : BOOL;
    knife5Lubrification     : BOOL;

    // Knife sharpening
    knife1Sharpening        : BOOL;
    knife2Sharpening        : BOOL;
    knife3Sharpening        : BOOL;
    knife4Sharpening        : BOOL;
    knife5Sharpening        : BOOL;

    knife1SharpeningLamp        : BOOL;
    knife2SharpeningLamp        : BOOL;
    knife3SharpeningLamp        : BOOL;
    knife4SharpeningLamp        : BOOL;
    knife5SharpeningLamp        : BOOL;	

	slitterCenterGuideRoll		: BOOL;

	
	rotaryKnifeInfeedUpperDamper1 : BOOL;
	rotaryKnifeInfeedUpperDamper2 : BOOL;
	
	rotaryKnifeInfeedLowerDamper1 : BOOL;
	rotaryKnifeInfeedLowerDamper2 : BOOL;
	
	pilotRollUpDown			: BOOL;	

    outfeedRoll_Up       : BOOL; // Raise the roll
    outfeedRoll_Down     : BOOL; // Lower the roll	
	
    // Paper direction flaps
    paperDirectionFlap01    : BOOL;
    paperDirectionFlap02    : BOOL;
    paperDirectionFlap03    : BOOL;
    paperDirectionFlap04    : BOOL;
    paperDirectionFlap05    : BOOL;
    paperDirectionFlap06    : BOOL;
    paperDirectionFlap07    : BOOL;
    paperDirectionFlap08    : BOOL;
    paperDirectionFlap09    : BOOL;
    paperDirectionFlap10    : BOOL;
    paperDirectionFlap11    : BOOL;
    paperDirectionFlap12    : BOOL;

    // Slitter movement controls
    moveSlitterOperatorSide : BOOL;
    moveSlitterMotorSide    : BOOL;
    moveSlitterOperatorSideLamp : BOOL;
    moveSlitterMotorSideLamp    : BOOL;	
	

    // Paper scrap controls
    paperTrimOperatorSideOpen  : BOOL;
    paperTrimOperatorSideClose : BOOL;
    paperTrimMotorSideOpen     : BOOL;
    paperTrimMotorSideClose    : BOOL;

	

	scorerHeightInc		: BOOL;	
	scorerHeightDec		: BOOL;	
	scorerHeightMotorStart : BOOL;
	scorerHeightMotorSlow : BOOL;
	scorerHeightMotorFast : BOOL;
	
	
	
	scorerTypeWLamp		: BOOL;
	scorerTypeNLamp		: BOOL;	
	scorerTypeDLamp		: BOOL;		
	
	
    // Motor commands
	tractionEnabledLamp		: BOOL;
    knifeMotorStart         : BOOL;
    scorerMotorStart        : BOOL;
	slitterKnifeDriveRef           : REAL;  // Knife motor start command / Partida motor facas	
    slitterScorerDriveRef          : REAL;  // Scorer motor start command / Partida motor vincos	
		
	
	startExhaustMotor				: BOOL;
	startExhaustMotorLamp			: BOOL;
	
	
	arrKnifeRunningMetersForSharpening		: ARRAY [1..5] OF INT;	(*This array is used to reset the lifetime meters that the knife runs*)
	arrKnifeRunningMetersForLubfrication		: ARRAY [1..5] OF INT;	(*This array is used to reset the lifetime meters that the knife runs*)
	
	hmiStatus				: slitterStatus_TypeStruct;
	
	
END_VAR

VAR PERSISTENT
	
	inst_FB_KnifeSharpening  : ARRAY [1..5] OF FB_KnifeSharpening;
	inst_FB_KnifeLubrification : ARRAY [1..5] OF	FB_KnifeLubrification;

END_VAR


VAR
    // Knife axis control instances
    instFB_AxisControlKnife1_Axis : FB_SimpleAxisControl;
    instFB_AxisControlKnife2_Axis : FB_SimpleAxisControl;
    instFB_AxisControlKnife3_Axis : FB_SimpleAxisControl;
    instFB_AxisControlKnife4_Axis : FB_SimpleAxisControl;
    instFB_AxisControlKnife5_Axis : FB_SimpleAxisControl;

    // Scorer axis control instances
    instFB_AxisControlScorer1_Axis : FB_SimpleAxisControl;
    instFB_AxisControlScorer2_Axis : FB_SimpleAxisControl;
    instFB_AxisControlScorer3_Axis : FB_SimpleAxisControl;
    instFB_AxisControlScorer4_Axis : FB_SimpleAxisControl;
    instFB_AxisControlScorer5_Axis : FB_SimpleAxisControl;
    instFB_AxisControlScorer6_Axis : FB_SimpleAxisControl;
    instFB_AxisControlScorer7_Axis : FB_SimpleAxisControl;
    instFB_AxisControlScorer8_Axis : FB_SimpleAxisControl;
    
    // Knife axis configurations
    knife1_AxisConfiguration : LAxisCtrl_typeAxisConfig;
    knife2_AxisConfiguration : LAxisCtrl_typeAxisConfig;
    knife3_AxisConfiguration : LAxisCtrl_typeAxisConfig;
    knife4_AxisConfiguration : LAxisCtrl_typeAxisConfig;
    knife5_AxisConfiguration : LAxisCtrl_typeAxisConfig;

    // Scorer axis configurations
    scorer1_AxisConfiguration : LAxisCtrl_typeAxisConfig;
    scorer2_AxisConfiguration : LAxisCtrl_typeAxisConfig;
    scorer3_AxisConfiguration : LAxisCtrl_typeAxisConfig;
    scorer4_AxisConfiguration : LAxisCtrl_typeAxisConfig;
    scorer5_AxisConfiguration : LAxisCtrl_typeAxisConfig;
    scorer6_AxisConfiguration : LAxisCtrl_typeAxisConfig;
    scorer7_AxisConfiguration : LAxisCtrl_typeAxisConfig;
    scorer8_AxisConfiguration : LAxisCtrl_typeAxisConfig;
    
    // Knife sharpening and lubrication instances
    instSharpeningKnifeArr  : ARRAY [1..20] OF FB_KnifeSharpening_old;
    instKnifeLubrificationArr : ARRAY [1..20] OF FB_KnifeLubrification;

    // Timers
    instSlitterMotoringTP   : TP;    // Slitter motoring stop timer
    instFbCurrentOrderPositionsGeneration : FB_PositionsGeneration;
    instFbToggleStartKnife  : TOGGLE;
    instFbTPStopKnifeMotor  : TP;
    instFbToggleStartScorer : TOGGLE;
    instFbTPStopScorerMotor : TP;
    instFbScorerHeight      : FB_ScorerHeight;
    instTonDelay            : TON;
    instTONExecutePositioningDelay : TON;
    instTPHaltAxis          : TP;

    // Positioning status
    positioningRunning                  : BOOL;
    positioningFinished                 : BOOL;
    innerScorerPositioningRunning       : BOOL;
    outerScorerPositioningRunning       : BOOL;
    knifePositioningRunning             : BOOL;
    innerScorerPositioningFinished      : BOOL;
    outerScorerPositioningFinished      : BOOL;
    knifePositioningFinished            : BOOL;

    // Error flags
    knifeAxisError                      : BOOL;
    innerScorerError                    : BOOL;
    outerScorerError                    : BOOL;
    positioningAxisError                 : BOOL;

    // Motor running flags
    knifeMotorRun                       : BOOL;
    scorerMotorRun                      : BOOL;

    // State tracking
    executePositioningOld               : BOOL;
    changeOrderOld                      : BOOL;
    executeHomeOld                      : BOOL;
    homeRunning                         : BOOL;
    positioningStarted                  : BOOL;
    haltAxis                            : BOOL;

    // Positioning range checks
    knifePositionSetpointOutOfRange     : BOOL;
    innerScorerPositionSetpointOutOfRange : BOOL;
    outerScorerPositionSetpointOutOfRange : BOOL;

    // Aux timers
    auxiliarTP1                         : TP;
	knife1EnabledCmdOld: BOOL;
	knife2EnabledCmdOld: BOOL;
	knife3EnabledCmdOld: BOOL;
	knife4EnabledCmdOld: BOOL;
	knife5EnabledCmdOld: BOOL;

	scorer1EnabledCmdOld: BOOL;
	scorer2EnabledCmdOld: BOOL;
	scorer3EnabledCmdOld: BOOL;
	scorer4EnabledCmdOld: BOOL;
	scorer5EnabledCmdOld: BOOL;
	scorer6EnabledCmdOld: BOOL;
	scorer7EnabledCmdOld: BOOL;
	scorer8EnabledCmdOld: BOOL;
	
	
	inTargetPosition: BOOL;
	
	scorerTypeWCmdOld	: BOOL;
	scorerTypeNCmdOld	: BOOL;	
	scorerTypeDCmdOld	: BOOL;	
	
	instKnifeSharpeningCLK_PRG: CLK_PRG;
	instKnifeLubrificationCLK_PRG: CLK_PRG;
	instTOFScorerSensorDelay: TOF;
	scorerHeightPositioningRunning: BOOL;
	scorerHeightPositioningState: INT;
	inst_GEN_PULSE_1S: GEN_PULSE;
	clock_Pulse_1S: BOOL;
	instFB_PaperDirectionControl : FB_PaperDirectionControl;	
	instRTrigToolsInPosition: R_TRIG;

	
	flapsSetAutoOld: BOOL;
	bAllKnivesInPos: BOOL;
	displayFlapsIndex: INT;
	displayKnifesIndex: INT;
	knifeRunningMetersArr: INT;
	outfeedRoll_DownCmdOld: BOOL;
	outfeedRoll_UpCmdOld: BOOL;
	instTONOutfeedRollDelay: TON;
	
	
	generatePositionsTest: BOOL;
	generatePositionsTestOld: BOOL;
END_VAR

VAR CONSTANT
    AXIS_TYPE_KNIFE         : INT := 1;
    AXIS_TYPE_INNER_SCORER  : INT := 2;
    AXIS_TYPE_OUTER_SCORER  : INT := 3;
END_VAR

(*Update axis status at the beginning of every cicle*)
knife1_Axis();
knife2_Axis();
knife3_Axis();
knife4_Axis();
knife5_Axis();

scorer1_Axis();
scorer2_Axis();
scorer3_Axis();
scorer4_Axis();
scorer5_Axis();
scorer6_Axis();
scorer7_Axis();
scorer8_Axis();

(*Update inverter status at the beginning of every cicle*)


(*Call program subroutines*)

_axisControl();
_toolsUpDownControl();
_slitterDisplacement();
//_knifeSharpening_old();
_knifeSharpening();

_paperTrim();
_safetyCircuit();
_startStopCutting();
_scorerHeightControl();
_exhaustMotor();
_startTractionMotor();
_knifeSharpening_old();
_knifeLubrification();
//_paperDirectionFlaps();
_slitterPaperDirectionControl();

_slitterCenterPaperGuideRoll();
_09_OutFeedRoll();

ACT_AlarmActive();
ACT_Alarms();
ACT_AuxiliaryCommands();
ACT_ProgramCurrentOrder();

ACT_GeneratePositions();
_haltTheAxis();
_homeFinished();
_08_HmiStatusDisplay();

_toolEnabledLamp();

EN := TRUE;

IF generatePositionsTest AND NOT generatePositionsTestOld THEN
	
	
	instFbCurrentOrderPositionsGeneration(execute := TRUE,
		machineConfig := machineConfig,
		currentOrder := currentOrder);
	
END_IF

generatePositionsTestOld := generatePositionsTest;

METHOD _08_HmiStatusDisplay


FOR displayFlapsIndex := 1 TO 27 DO
	
	
	hmiStatus.flapSolenoidArr[displayFlapsIndex] :=	instFB_PaperDirectionControl.flapSolenoidArr[displayFlapsIndex];

END_FOR


FOR displayKnifesIndex := 1 TO 5 DO
	
	
	hmiStatus.knifeRunningMetersArr[displayKnifesIndex] := inst_FB_KnifeSharpening[displayKnifesIndex].knifeRunningMeters;
	hmiStatus.knifeRunningMetersTotalArr[displayKnifesIndex] := inst_FB_KnifeSharpening[displayKnifesIndex].knifeRunningMetersTotal;
	
	hmiStatus.lubrificationRunningMetersArr[displayKnifesIndex] := inst_FB_KnifeLubrification[displayKnifesIndex].knifeRunningMeters;
	
	
END_FOR
END_METHOD

METHOD _09_OutFeedRoll : BOOL
// ==========================================================================
// OUTFEED ROLL CONTROL LOGIC
// Location: Slitter Scorer Outfeed (Cardboard)
// ==========================================================================

// Update delay timer for automatic paper detection
instTONOutfeedRollDelay(IN := paperPresenceSensor, PT := T#15S);

// Logic Calculation Section
IF outfeedRoll_ManCmd THEN
    
    // Manual Toggle: Raise roll on rising edge of Up command
    IF outfeedRoll_UpCmd AND NOT outfeedRoll_UpCmdOld THEN
        outfeedRoll_Up   := TRUE;
        outfeedRoll_Down := FALSE;
    END_IF
    
    // Manual Toggle: Lower roll on rising edge of Down command
    IF outfeedRoll_DownCmd AND NOT outfeedRoll_DownCmdOld THEN
        outfeedRoll_Up   := FALSE;
        outfeedRoll_Down := TRUE;
    END_IF	

ELSE
    // AUTOMATIC MODE
    // Lower roll only if paper is present and the stable-presence delay has expired
    IF paperPresenceSensor AND instTONOutfeedRollDelay.Q THEN
        outfeedRoll_Up   := FALSE;
        outfeedRoll_Down := TRUE;
    ELSE
        // Default position: Keep roll raised
        outfeedRoll_Up   := TRUE;
        outfeedRoll_Down := FALSE;
    END_IF	

END_IF

// ==========================================================================
// SAFETY INTERLOCK & OUTPUT MAPPING
// ==========================================================================
// If safety feedback is lost, force both outputs to FALSE (Disable Movement)
IF NOT safetyFeedback THEN
    outfeedRoll_Up   := FALSE;
    outfeedRoll_Down := FALSE;
END_IF

// Store states for manual edge detection in next scan cycle
outfeedRoll_UpCmdOld   := outfeedRoll_UpCmd;
outfeedRoll_DownCmdOld := outfeedRoll_DownCmd;
END_METHOD

METHOD _axisControl
VAR_INPUT
END_VAR
(*

	limitSensorKnife3_4					: BOOL;
	limitSensorScorer4_6					: BOOL;
	limitSensorScorer3_5					: BOOL;
*)
(*==============================================================================================================================
Improved Knife Homing Sequence - CPNTeck Automation
===============================================================================================================================*)

(* Detect rising edge of executeHome *)
IF executeHome AND NOT executeHomeOld THEN
    homeRunning := TRUE;
    instTonDelay(IN := FALSE); // Reset timer
END_IF
executeHomeOld := executeHome;

(* Main Homing Logic *)
IF homeRunning THEN
    instTonDelay(IN := TRUE, PT := T#60S); // Start the 10s timer

    // Start homing Knife 1 and 5 after 1ms
    IF instTonDelay.ET > T#0S AND instTonDelay.ET <= T#10S THEN
        instFB_AxisControlKnife1_Axis.homing := TRUE;
        instFB_AxisControlKnife5_Axis.homing := TRUE;
		
		instFB_AxisControlScorer1_Axis.homing := TRUE;
		instFB_AxisControlScorer7_Axis.homing := TRUE;
		instFB_AxisControlScorer2_Axis.homing := TRUE;
		instFB_AxisControlScorer8_Axis.homing := TRUE;
		
		
    END_IF

    // Start homing Knife 2 and 4 after 3s
    IF instTonDelay.ET > T#10S AND instTonDelay.ET <= T#20S THEN
        instFB_AxisControlKnife2_Axis.homing := TRUE;
        instFB_AxisControlKnife4_Axis.homing := TRUE;
		
		instFB_AxisControlScorer4_Axis.homing := TRUE;
		instFB_AxisControlScorer6_Axis.homing := TRUE;
		instFB_AxisControlScorer3_Axis.homing := TRUE;
		instFB_AxisControlScorer5_Axis.homing := TRUE;
		
    END_IF

    // Start homing Knife 3 after 6s
    IF instTonDelay.ET > T#30S THEN
        instFB_AxisControlKnife3_Axis.homing := TRUE;
    END_IF

    // Finish sequence when timer completes
    IF instTonDelay.Q THEN
        homeRunning := FALSE;

        (* Reset all homing commands *)
        instFB_AxisControlKnife1_Axis.homing := FALSE;
        instFB_AxisControlKnife2_Axis.homing := FALSE;
        instFB_AxisControlKnife3_Axis.homing := FALSE;
        instFB_AxisControlKnife4_Axis.homing := FALSE;
        instFB_AxisControlKnife5_Axis.homing := FALSE;
		
		instFB_AxisControlScorer1_Axis.homing := FALSE;
		instFB_AxisControlScorer2_Axis.homing := FALSE;
		instFB_AxisControlScorer3_Axis.homing := FALSE;
		instFB_AxisControlScorer4_Axis.homing := FALSE;
		instFB_AxisControlScorer5_Axis.homing := FALSE;
		instFB_AxisControlScorer6_Axis.homing := FALSE;
		instFB_AxisControlScorer7_Axis.homing := FALSE;
		instFB_AxisControlScorer8_Axis.homing := FALSE;

        instTonDelay(IN := FALSE); // Stop the timer
    END_IF

ELSE
(*	
    (* Not running, ensure homing off and timer stopped *)
    instFB_AxisControlKnife1_Axis.homing := FALSE;
    instFB_AxisControlKnife2_Axis.homing := FALSE;
    instFB_AxisControlKnife3_Axis.homing := FALSE;
    instFB_AxisControlKnife4_Axis.homing := FALSE;
    instFB_AxisControlKnife5_Axis.homing := FALSE;
	
	instFB_AxisControlScorer1_Axis.homing := FALSE;
	instFB_AxisControlScorer2_Axis.homing := FALSE;
	instFB_AxisControlScorer3_Axis.homing := FALSE;
	instFB_AxisControlScorer4_Axis.homing := FALSE;
	instFB_AxisControlScorer5_Axis.homing := FALSE;
	instFB_AxisControlScorer6_Axis.homing := FALSE;
	instFB_AxisControlScorer7_Axis.homing := FALSE;
	instFB_AxisControlScorer8_Axis.homing := FALSE;	
    instTonDelay(IN := FALSE);
*)	
END_IF
//----------------------------------------------------------------------------------------------
// Knife Axis parameters setup
//----------------------------------------------------------------------------------------------

//Knife 1 - Axis home parameters
knife1_AxisConfiguration.homing.position := machineConfig.homePositionKnife[1];
knife1_AxisConfiguration.homing.offsetPosition := machineConfig.homePositionKnife[1];
knife1_AxisConfiguration.homing.homeExecutionTimeLimit := T#5M;

//Knife 1 - Axis positioning abosulute parameters
knife1_AxisConfiguration.posAbsolute.position := currentOrder.generatedOrder.knifePositionReferenceArr[1] + machineConfig.knifePositionCorrectionArr[1];
knife1_AxisConfiguration.posAbsolute.velocity := machineConfig.toolFastPositioningVelocity;
knife1_AxisConfiguration.posAbsolute.acceleration := machineConfig.toolFastPositioningAccel;
knife1_AxisConfiguration.posAbsolute.deceleration := machineConfig.toolFastPositioningDecel;
knife1_AxisConfiguration.posAbsolute.jerk := machineConfig.toolFastPositioningJerk;


//Knife 1 - Axis positioning relative parameters
knife1_AxisConfiguration.posRelative.distance := hmiCommands.slitter1.knifePosCorrectionArr[1].positionCorrection;
knife1_AxisConfiguration.posRelative.direction := 0;
knife1_AxisConfiguration.posRelative.velocity := machineConfig.toolSlowPositioningVelocity;
knife1_AxisConfiguration.posRelative.acceleration := machineConfig.toolSlowPositioningAccel;
knife1_AxisConfiguration.posRelative.deceleration := machineConfig.toolFastPositioningAccel;
knife1_AxisConfiguration.posRelative.jerk := machineConfig.toolSlowPositioningJerk;

//Knife 1 - Axis JOG parameters
knife1_AxisConfiguration.jog.velocity := machineConfig.toolSlowPositioningVelocity;
knife1_AxisConfiguration.jog.acceleration := machineConfig.toolSlowPositioningAccel;
knife1_AxisConfiguration.jog.deceleration := machineConfig.toolFastPositioningAccel;
knife1_AxisConfiguration.jog.jerk := machineConfig.toolSlowPositioningJerk;



//Knife 2
knife2_AxisConfiguration.homing.position := machineConfig.homePositionKnife[2];
knife2_AxisConfiguration.homing.offsetPosition := machineConfig.homePositionKnife[2];
knife2_AxisConfiguration.homing.homeExecutionTimeLimit := T#5M;

knife2_AxisConfiguration.posAbsolute.position := currentOrder.generatedOrder.knifePositionReferenceArr[2] + machineConfig.knifePositionCorrectionArr[2];
knife2_AxisConfiguration.posAbsolute.velocity := machineConfig.toolFastPositioningVelocity;
knife2_AxisConfiguration.posAbsolute.acceleration := machineConfig.toolFastPositioningAccel;
knife2_AxisConfiguration.posAbsolute.deceleration := machineConfig.toolFastPositioningDecel;
knife2_AxisConfiguration.posAbsolute.jerk := machineConfig.toolFastPositioningJerk;


//Knife 2 - Axis positioning relative parameters
knife2_AxisConfiguration.posRelative.distance := hmiCommands.slitter1.knifePosCorrectionArr[2].positionCorrection;
knife2_AxisConfiguration.posRelative.direction := 0;
knife2_AxisConfiguration.posRelative.velocity := machineConfig.toolSlowPositioningVelocity;
knife2_AxisConfiguration.posRelative.acceleration := machineConfig.toolSlowPositioningAccel;
knife2_AxisConfiguration.posRelative.deceleration := machineConfig.toolFastPositioningAccel;
knife2_AxisConfiguration.posRelative.jerk := machineConfig.toolSlowPositioningJerk;

//Knife 2 - Axis JOG parameters
knife2_AxisConfiguration.jog.velocity := machineConfig.toolSlowPositioningVelocity;
knife2_AxisConfiguration.jog.acceleration := machineConfig.toolSlowPositioningAccel;
knife2_AxisConfiguration.jog.deceleration := machineConfig.toolFastPositioningAccel;
knife2_AxisConfiguration.jog.jerk := machineConfig.toolSlowPositioningJerk;



//Knife 3
knife3_AxisConfiguration.homing.position := machineConfig.homePositionKnife[3];
knife3_AxisConfiguration.homing.offsetPosition :=  machineConfig.homePositionKnife[3];
knife3_AxisConfiguration.homing.homeExecutionTimeLimit := T#5M;

knife3_AxisConfiguration.posAbsolute.position := currentOrder.generatedOrder.knifePositionReferenceArr[3] + machineConfig.knifePositionCorrectionArr[3];
knife3_AxisConfiguration.posAbsolute.velocity := machineConfig.toolFastPositioningVelocity;
knife3_AxisConfiguration.posAbsolute.acceleration := machineConfig.toolFastPositioningAccel;
knife3_AxisConfiguration.posAbsolute.deceleration := machineConfig.toolFastPositioningDecel;
knife3_AxisConfiguration.posAbsolute.jerk := machineConfig.toolFastPositioningJerk;


//Knife 3 - Axis positioning relative parameters
knife3_AxisConfiguration.posRelative.distance := hmiCommands.slitter1.knifePosCorrectionArr[3].positionCorrection;
knife3_AxisConfiguration.posRelative.direction := 0;
knife3_AxisConfiguration.posRelative.velocity := machineConfig.toolSlowPositioningVelocity;
knife3_AxisConfiguration.posRelative.acceleration := machineConfig.toolSlowPositioningAccel;
knife3_AxisConfiguration.posRelative.deceleration := machineConfig.toolFastPositioningAccel;
knife3_AxisConfiguration.posRelative.jerk := machineConfig.toolSlowPositioningJerk;

//Knife 3 - Axis JOG parameters
knife3_AxisConfiguration.jog.velocity := machineConfig.toolSlowPositioningVelocity;
knife3_AxisConfiguration.jog.acceleration := machineConfig.toolSlowPositioningAccel;
knife3_AxisConfiguration.jog.deceleration := machineConfig.toolFastPositioningAccel;
knife3_AxisConfiguration.jog.jerk := machineConfig.toolSlowPositioningJerk;



//Knife 4
knife4_AxisConfiguration.homing.position := machineConfig.homePositionKnife[4];
knife4_AxisConfiguration.homing.offsetPosition :=  machineConfig.homePositionKnife[4];
knife4_AxisConfiguration.homing.homeExecutionTimeLimit := T#5M;

knife4_AxisConfiguration.posAbsolute.position := currentOrder.generatedOrder.knifePositionReferenceArr[4] + machineConfig.knifePositionCorrectionArr[4];
knife4_AxisConfiguration.posAbsolute.velocity := machineConfig.toolFastPositioningVelocity;
knife4_AxisConfiguration.posAbsolute.acceleration := machineConfig.toolFastPositioningAccel;
knife4_AxisConfiguration.posAbsolute.deceleration := machineConfig.toolFastPositioningDecel;
knife4_AxisConfiguration.posAbsolute.jerk := machineConfig.toolFastPositioningJerk;


//Knife 4 - Axis positioning relative parameters
knife4_AxisConfiguration.posRelative.distance := hmiCommands.slitter1.knifePosCorrectionArr[4].positionCorrection;
knife4_AxisConfiguration.posRelative.direction := 0;
knife4_AxisConfiguration.posRelative.velocity := machineConfig.toolSlowPositioningVelocity;
knife4_AxisConfiguration.posRelative.acceleration := machineConfig.toolSlowPositioningAccel;
knife4_AxisConfiguration.posRelative.deceleration := machineConfig.toolFastPositioningAccel;
knife4_AxisConfiguration.posRelative.jerk := machineConfig.toolSlowPositioningJerk;

//Knife 4 - Axis JOG parameters
knife4_AxisConfiguration.jog.velocity := machineConfig.toolSlowPositioningVelocity;
knife4_AxisConfiguration.jog.acceleration := machineConfig.toolSlowPositioningAccel;
knife4_AxisConfiguration.jog.deceleration := machineConfig.toolFastPositioningAccel;
knife4_AxisConfiguration.jog.jerk := machineConfig.toolSlowPositioningJerk;


//Knife 5
knife5_AxisConfiguration.homing.position := machineConfig.homePositionKnife[5];
knife5_AxisConfiguration.homing.offsetPosition :=  machineConfig.homePositionKnife[5];
knife5_AxisConfiguration.homing.homeExecutionTimeLimit := T#5M;

knife5_AxisConfiguration.posAbsolute.position := currentOrder.generatedOrder.knifePositionReferenceArr[5] + machineConfig.knifePositionCorrectionArr[5];
knife5_AxisConfiguration.posAbsolute.velocity := machineConfig.toolFastPositioningVelocity;
knife5_AxisConfiguration.posAbsolute.acceleration := machineConfig.toolFastPositioningAccel;
knife5_AxisConfiguration.posAbsolute.deceleration := machineConfig.toolFastPositioningDecel;
knife5_AxisConfiguration.posAbsolute.jerk := machineConfig.toolFastPositioningJerk;

//Knife 5 - Axis positioning relative parameters
knife5_AxisConfiguration.posRelative.distance := hmiCommands.slitter1.knifePosCorrectionArr[5].positionCorrection;
knife5_AxisConfiguration.posRelative.direction := 0;
knife5_AxisConfiguration.posRelative.velocity := machineConfig.toolSlowPositioningVelocity;
knife5_AxisConfiguration.posRelative.acceleration := machineConfig.toolSlowPositioningAccel;
knife5_AxisConfiguration.posRelative.deceleration := machineConfig.toolFastPositioningAccel;
knife5_AxisConfiguration.posRelative.jerk := machineConfig.toolSlowPositioningJerk;

//Knife 5 - Axis JOG parameters
knife5_AxisConfiguration.jog.velocity := machineConfig.toolSlowPositioningVelocity;
knife5_AxisConfiguration.jog.acceleration := machineConfig.toolSlowPositioningAccel;
knife5_AxisConfiguration.jog.deceleration := machineConfig.toolFastPositioningAccel;
knife5_AxisConfiguration.jog.jerk := machineConfig.toolSlowPositioningJerk;


//----------------------------------------------------------------------------------------------
// Scorer Axis parameters setup
//----------------------------------------------------------------------------------------------

//Scorer 1
scorer1_AxisConfiguration.homing.position := machineConfig.homePositionScorer[1];
scorer1_AxisConfiguration.homing.offsetPosition := machineConfig.homePositionScorer[1];
scorer1_AxisConfiguration.homing.homeExecutionTimeLimit := T#5M;

scorer1_AxisConfiguration.posAbsolute.position := currentOrder.generatedOrder.scorerPositionReferenceArr[1] + machineConfig.scorerPositionCorrectionArr[1];
scorer1_AxisConfiguration.posAbsolute.velocity := machineConfig.toolFastPositioningVelocity;
scorer1_AxisConfiguration.posAbsolute.acceleration := machineConfig.toolFastPositioningAccel;
scorer1_AxisConfiguration.posAbsolute.deceleration := machineConfig.toolFastPositioningDecel;
scorer1_AxisConfiguration.posAbsolute.jerk := machineConfig.toolFastPositioningJerk;

//Scorer 1 - Axis positioning relative parameters
scorer1_AxisConfiguration.posRelative.distance := hmiCommands.slitter1.scorerPosCorrectionArr[1].positionCorrection;
scorer1_AxisConfiguration.posRelative.direction := 0;
scorer1_AxisConfiguration.posRelative.velocity := machineConfig.toolSlowPositioningVelocity;
scorer1_AxisConfiguration.posRelative.acceleration := machineConfig.toolSlowPositioningAccel;
scorer1_AxisConfiguration.posRelative.deceleration := machineConfig.toolFastPositioningAccel;
scorer1_AxisConfiguration.posRelative.jerk := machineConfig.toolSlowPositioningJerk;

//Scorer 1 - Axis JOG parameters
scorer1_AxisConfiguration.jog.velocity := machineConfig.toolSlowPositioningVelocity;
scorer1_AxisConfiguration.jog.acceleration := machineConfig.toolSlowPositioningAccel;
scorer1_AxisConfiguration.jog.deceleration := machineConfig.toolFastPositioningAccel;
scorer1_AxisConfiguration.jog.jerk := machineConfig.toolSlowPositioningJerk;


//Scorer 2
scorer2_AxisConfiguration.homing.position := machineConfig.homePositionScorer[2];
scorer2_AxisConfiguration.homing.offsetPosition := machineConfig.homePositionScorer[2];
scorer2_AxisConfiguration.homing.homeExecutionTimeLimit := T#5M;

scorer2_AxisConfiguration.posAbsolute.position := currentOrder.generatedOrder.scorerPositionReferenceArr[2] + machineConfig.scorerPositionCorrectionArr[2];
scorer2_AxisConfiguration.posAbsolute.velocity := machineConfig.toolFastPositioningVelocity;
scorer2_AxisConfiguration.posAbsolute.acceleration := machineConfig.toolFastPositioningAccel;
scorer2_AxisConfiguration.posAbsolute.deceleration := machineConfig.toolFastPositioningDecel;
scorer2_AxisConfiguration.posAbsolute.jerk := machineConfig.toolFastPositioningJerk;

//Scorer 2 - Axis positioning relative parameters
scorer2_AxisConfiguration.posRelative.distance := hmiCommands.slitter1.scorerPosCorrectionArr[2].positionCorrection;
scorer2_AxisConfiguration.posRelative.direction := 0;
scorer2_AxisConfiguration.posRelative.velocity := machineConfig.toolSlowPositioningVelocity;
scorer2_AxisConfiguration.posRelative.acceleration := machineConfig.toolSlowPositioningAccel;
scorer2_AxisConfiguration.posRelative.deceleration := machineConfig.toolFastPositioningAccel;
scorer2_AxisConfiguration.posRelative.jerk := machineConfig.toolSlowPositioningJerk;

//Scorer 2 - Axis JOG parameters
scorer2_AxisConfiguration.jog.velocity := machineConfig.toolSlowPositioningVelocity;
scorer2_AxisConfiguration.jog.acceleration := machineConfig.toolSlowPositioningAccel;
scorer2_AxisConfiguration.jog.deceleration := machineConfig.toolFastPositioningAccel;
scorer2_AxisConfiguration.jog.jerk := machineConfig.toolSlowPositioningJerk;

//Scorer 3
scorer3_AxisConfiguration.homing.position := machineConfig.homePositionScorer[3];
scorer3_AxisConfiguration.homing.offsetPosition := machineConfig.homePositionScorer[3];
scorer3_AxisConfiguration.homing.homeExecutionTimeLimit := T#5M;

scorer3_AxisConfiguration.posAbsolute.position := currentOrder.generatedOrder.scorerPositionReferenceArr[3] + machineConfig.scorerPositionCorrectionArr[3];
scorer3_AxisConfiguration.posAbsolute.velocity := machineConfig.toolFastPositioningVelocity;
scorer3_AxisConfiguration.posAbsolute.acceleration := machineConfig.toolFastPositioningAccel;
scorer3_AxisConfiguration.posAbsolute.deceleration := machineConfig.toolFastPositioningDecel;
scorer3_AxisConfiguration.posAbsolute.jerk := machineConfig.toolFastPositioningJerk;

//Scorer 3 - Axis positioning relative parameters
scorer3_AxisConfiguration.posRelative.distance := hmiCommands.slitter1.scorerPosCorrectionArr[3].positionCorrection;
scorer3_AxisConfiguration.posRelative.direction := 0;
scorer3_AxisConfiguration.posRelative.velocity := machineConfig.toolSlowPositioningVelocity;
scorer3_AxisConfiguration.posRelative.acceleration := machineConfig.toolSlowPositioningAccel;
scorer3_AxisConfiguration.posRelative.deceleration := machineConfig.toolFastPositioningAccel;
scorer3_AxisConfiguration.posRelative.jerk := machineConfig.toolSlowPositioningJerk;

//Scorer 3 - Axis JOG parameters
scorer3_AxisConfiguration.jog.velocity := machineConfig.toolSlowPositioningVelocity;
scorer3_AxisConfiguration.jog.acceleration := machineConfig.toolSlowPositioningAccel;
scorer3_AxisConfiguration.jog.deceleration := machineConfig.toolFastPositioningAccel;
scorer3_AxisConfiguration.jog.jerk := machineConfig.toolSlowPositioningJerk;



//Scorer 4
scorer4_AxisConfiguration.homing.position := machineConfig.homePositionScorer[4];
scorer4_AxisConfiguration.homing.offsetPosition := machineConfig.homePositionScorer[4];
scorer4_AxisConfiguration.homing.homeExecutionTimeLimit := T#5M;

scorer4_AxisConfiguration.posAbsolute.position := currentOrder.generatedOrder.scorerPositionReferenceArr[4] + machineConfig.scorerPositionCorrectionArr[4];
scorer4_AxisConfiguration.posAbsolute.velocity := machineConfig.toolFastPositioningVelocity;
scorer4_AxisConfiguration.posAbsolute.acceleration := machineConfig.toolFastPositioningAccel;
scorer4_AxisConfiguration.posAbsolute.deceleration := machineConfig.toolFastPositioningDecel;
scorer4_AxisConfiguration.posAbsolute.jerk := machineConfig.toolFastPositioningJerk;

//Scorer 4 - Axis positioning relative parameters
scorer4_AxisConfiguration.posRelative.distance := hmiCommands.slitter1.scorerPosCorrectionArr[4].positionCorrection;
scorer4_AxisConfiguration.posRelative.direction := 0;
scorer4_AxisConfiguration.posRelative.velocity := machineConfig.toolSlowPositioningVelocity;
scorer4_AxisConfiguration.posRelative.acceleration := machineConfig.toolSlowPositioningAccel;
scorer4_AxisConfiguration.posRelative.deceleration := machineConfig.toolFastPositioningAccel;
scorer4_AxisConfiguration.posRelative.jerk := machineConfig.toolSlowPositioningJerk;

//Scorer 4 - Axis JOG parameters
scorer4_AxisConfiguration.jog.velocity := machineConfig.toolSlowPositioningVelocity;
scorer4_AxisConfiguration.jog.acceleration := machineConfig.toolSlowPositioningAccel;
scorer4_AxisConfiguration.jog.deceleration := machineConfig.toolFastPositioningAccel;
scorer4_AxisConfiguration.jog.jerk := machineConfig.toolSlowPositioningJerk;



//Scorer 5
//_________________________________________________________________________________________________________________________
scorer5_AxisConfiguration.homing.position := machineConfig.homePositionScorer[5];
scorer5_AxisConfiguration.homing.offsetPosition := machineConfig.homePositionScorer[5];
scorer5_AxisConfiguration.homing.homeExecutionTimeLimit := T#5M;

scorer5_AxisConfiguration.posAbsolute.position := currentOrder.generatedOrder.scorerPositionReferenceArr[5] + machineConfig.scorerPositionCorrectionArr[5];
scorer5_AxisConfiguration.posAbsolute.velocity := machineConfig.toolFastPositioningVelocity;
scorer5_AxisConfiguration.posAbsolute.acceleration := machineConfig.toolFastPositioningAccel;
scorer5_AxisConfiguration.posAbsolute.deceleration := machineConfig.toolFastPositioningDecel;
scorer5_AxisConfiguration.posAbsolute.jerk := machineConfig.toolFastPositioningJerk;

//Scorer 5 - Axis positioning relative parameters
scorer5_AxisConfiguration.posRelative.distance := hmiCommands.slitter1.scorerPosCorrectionArr[5].positionCorrection;
scorer5_AxisConfiguration.posRelative.direction := 0;
scorer5_AxisConfiguration.posRelative.velocity := machineConfig.toolSlowPositioningVelocity;
scorer5_AxisConfiguration.posRelative.acceleration := machineConfig.toolSlowPositioningAccel;
scorer5_AxisConfiguration.posRelative.deceleration := machineConfig.toolFastPositioningAccel;
scorer5_AxisConfiguration.posRelative.jerk := machineConfig.toolSlowPositioningJerk;

//Scorer 5 - Axis JOG parameters
scorer5_AxisConfiguration.jog.velocity := machineConfig.toolSlowPositioningVelocity;
scorer5_AxisConfiguration.jog.acceleration := machineConfig.toolSlowPositioningAccel;
scorer5_AxisConfiguration.jog.deceleration := machineConfig.toolFastPositioningAccel;
scorer5_AxisConfiguration.jog.jerk := machineConfig.toolSlowPositioningJerk;

//Scorer 6
//_________________________________________________________________________________________________________________________
scorer6_AxisConfiguration.homing.position := machineConfig.homePositionScorer[6];
scorer6_AxisConfiguration.homing.offsetPosition := machineConfig.homePositionScorer[6];
scorer6_AxisConfiguration.homing.homeExecutionTimeLimit := T#5M;

scorer6_AxisConfiguration.posAbsolute.position := currentOrder.generatedOrder.scorerPositionReferenceArr[6] + machineConfig.scorerPositionCorrectionArr[6];
scorer6_AxisConfiguration.posAbsolute.velocity := machineConfig.toolFastPositioningVelocity;
scorer6_AxisConfiguration.posAbsolute.acceleration := machineConfig.toolFastPositioningAccel;
scorer6_AxisConfiguration.posAbsolute.deceleration := machineConfig.toolFastPositioningDecel;
scorer6_AxisConfiguration.posAbsolute.jerk := machineConfig.toolFastPositioningJerk;

//Scorer 6 - Axis positioning relative parameters
scorer6_AxisConfiguration.posRelative.distance := hmiCommands.slitter1.scorerPosCorrectionArr[6].positionCorrection;
scorer6_AxisConfiguration.posRelative.direction := 0;
scorer6_AxisConfiguration.posRelative.velocity := machineConfig.toolSlowPositioningVelocity;
scorer6_AxisConfiguration.posRelative.acceleration := machineConfig.toolSlowPositioningAccel;
scorer6_AxisConfiguration.posRelative.deceleration := machineConfig.toolFastPositioningAccel;
scorer6_AxisConfiguration.posRelative.jerk := machineConfig.toolSlowPositioningJerk;

//Scorer 6 - Axis JOG parameters
scorer6_AxisConfiguration.jog.velocity := machineConfig.toolSlowPositioningVelocity;
scorer6_AxisConfiguration.jog.acceleration := machineConfig.toolSlowPositioningAccel;
scorer6_AxisConfiguration.jog.deceleration := machineConfig.toolFastPositioningAccel;
scorer6_AxisConfiguration.jog.jerk := machineConfig.toolSlowPositioningJerk;

//Scorer 7
//_________________________________________________________________________________________________________________________

scorer7_AxisConfiguration.homing.position := machineConfig.homePositionScorer[7];
scorer7_AxisConfiguration.homing.offsetPosition := machineConfig.homePositionScorer[7];
scorer7_AxisConfiguration.homing.homeExecutionTimeLimit := T#5M;

scorer7_AxisConfiguration.posAbsolute.position := currentOrder.generatedOrder.scorerPositionReferenceArr[7] + machineConfig.scorerPositionCorrectionArr[7];
scorer7_AxisConfiguration.posAbsolute.velocity := machineConfig.toolFastPositioningVelocity;
scorer7_AxisConfiguration.posAbsolute.acceleration := machineConfig.toolFastPositioningAccel;
scorer7_AxisConfiguration.posAbsolute.deceleration := machineConfig.toolFastPositioningDecel;
scorer7_AxisConfiguration.posAbsolute.jerk := machineConfig.toolFastPositioningJerk;

